(* Logix 5000 project; controller TBEN_Lx_8IOL_AOI_V0_2 vendor 1 type 14 code 176 rev 32.11; software revision 32.00; part 5 of 16 *)

           TBEN_L4_8IOL:O.Data[63].0   // IO-Link Port 4 - Output data word 13 (INT bit0)
           TBEN_L4_8IOL:O.Data[63].1   // IO-Link Port 4 - Output data word 13 (INT bit1)
           TBEN_L4_8IOL:O.Data[63].10   // IO-Link Port 4 - Output data word 13 (INT bit10)
           TBEN_L4_8IOL:O.Data[63].11   // IO-Link Port 4 - Output data word 13 (INT bit11)
           TBEN_L4_8IOL:O.Data[63].12   // IO-Link Port 4 - Output data word 13 (INT bit12)
           TBEN_L4_8IOL:O.Data[63].13   // IO-Link Port 4 - Output data word 13 (INT bit13)
           TBEN_L4_8IOL:O.Data[63].14   // IO-Link Port 4 - Output data word 13 (INT bit14)
           TBEN_L4_8IOL:O.Data[63].15   // IO-Link Port 4 - Output data word 13 (INT bit15)
           TBEN_L4_8IOL:O.Data[63].2   // IO-Link Port 4 - Output data word 13 (INT bit2)
           TBEN_L4_8IOL:O.Data[63].3   // IO-Link Port 4 - Output data word 13 (INT bit3)
           TBEN_L4_8IOL:O.Data[63].4   // IO-Link Port 4 - Output data word 13 (INT bit4)
           TBEN_L4_8IOL:O.Data[63].5   // IO-Link Port 4 - Output data word 13 (INT bit5)
           TBEN_L4_8IOL:O.Data[63].6   // IO-Link Port 4 - Output data word 13 (INT bit6)
           TBEN_L4_8IOL:O.Data[63].7   // IO-Link Port 4 - Output data word 13 (INT bit7)
           TBEN_L4_8IOL:O.Data[63].8   // IO-Link Port 4 - Output data word 13 (INT bit8)
           TBEN_L4_8IOL:O.Data[63].9   // IO-Link Port 4 - Output data word 13 (INT bit9)
           TBEN_L4_8IOL:O.Data[64]   // IO-Link Port 4 - Output data word 14
           TBEN_L4_8IOL:O.Data[64].0   // IO-Link Port 4 - Output data word 14 (INT bit0)
           TBEN_L4_8IOL:O.Data[64].1   // IO-Link Port 4 - Output data word 14 (INT bit1)
           TBEN_L4_8IOL:O.Data[64].10   // IO-Link Port 4 - Output data word 14 (INT bit10)
           TBEN_L4_8IOL:O.Data[64].11   // IO-Link Port 4 - Output data word 14 (INT bit11)
           TBEN_L4_8IOL:O.Data[64].12   // IO-Link Port 4 - Output data word 14 (INT bit12)
           TBEN_L4_8IOL:O.Data[64].13   // IO-Link Port 4 - Output data word 14 (INT bit13)
           TBEN_L4_8IOL:O.Data[64].14   // IO-Link Port 4 - Output data word 14 (INT bit14)
           TBEN_L4_8IOL:O.Data[64].15   // IO-Link Port 4 - Output data word 14 (INT bit15)
           TBEN_L4_8IOL:O.Data[64].2   // IO-Link Port 4 - Output data word 14 (INT bit2)
           TBEN_L4_8IOL:O.Data[64].3   // IO-Link Port 4 - Output data word 14 (INT bit3)
           TBEN_L4_8IOL:O.Data[64].4   // IO-Link Port 4 - Output data word 14 (INT bit4)
           TBEN_L4_8IOL:O.Data[64].5   // IO-Link Port 4 - Output data word 14 (INT bit5)
           TBEN_L4_8IOL:O.Data[64].6   // IO-Link Port 4 - Output data word 14 (INT bit6)
           TBEN_L4_8IOL:O.Data[64].7   // IO-Link Port 4 - Output data word 14 (INT bit7)
           TBEN_L4_8IOL:O.Data[64].8   // IO-Link Port 4 - Output data word 14 (INT bit8)
           TBEN_L4_8IOL:O.Data[64].9   // IO-Link Port 4 - Output data word 14 (INT bit9)
           TBEN_L4_8IOL:O.Data[65]   // IO-Link Port 4 - Output data word 15
           TBEN_L4_8IOL:O.Data[65].0   // IO-Link Port 4 - Output data word 15 (INT bit0)
           TBEN_L4_8IOL:O.Data[65].1   // IO-Link Port 4 - Output data word 15 (INT bit1)
           TBEN_L4_8IOL:O.Data[65].10   // IO-Link Port 4 - Output data word 15 (INT bit10)
           TBEN_L4_8IOL:O.Data[65].11   // IO-Link Port 4 - Output data word 15 (INT bit11)
           TBEN_L4_8IOL:O.Data[65].12   // IO-Link Port 4 - Output data word 15 (INT bit12)
           TBEN_L4_8IOL:O.Data[65].13   // IO-Link Port 4 - Output data word 15 (INT bit13)
           TBEN_L4_8IOL:O.Data[65].14   // IO-Link Port 4 - Output data word 15 (INT bit14)
           TBEN_L4_8IOL:O.Data[65].15   // IO-Link Port 4 - Output data word 15 (INT bit15)
           TBEN_L4_8IOL:O.Data[65].2   // IO-Link Port 4 - Output data word 15 (INT bit2)
           TBEN_L4_8IOL:O.Data[65].3   // IO-Link Port 4 - Output data word 15 (INT bit3)
           TBEN_L4_8IOL:O.Data[65].4   // IO-Link Port 4 - Output data word 15 (INT bit4)
           TBEN_L4_8IOL:O.Data[65].5   // IO-Link Port 4 - Output data word 15 (INT bit5)
           TBEN_L4_8IOL:O.Data[65].6   // IO-Link Port 4 - Output data word 15 (INT bit6)
           TBEN_L4_8IOL:O.Data[65].7   // IO-Link Port 4 - Output data word 15 (INT bit7)
           TBEN_L4_8IOL:O.Data[65].8   // IO-Link Port 4 - Output data word 15 (INT bit8)
           TBEN_L4_8IOL:O.Data[65].9   // IO-Link Port 4 - Output data word 15 (INT bit9)
           TBEN_L4_8IOL:O.Data[66]   // IO-Link Port 5 - Output data word 0
           TBEN_L4_8IOL:O.Data[66].0   // IO-Link Port 5 - Output data word 0 (INT bit0)
           TBEN_L4_8IOL:O.Data[66].1   // IO-Link Port 5 - Output data word 0 (INT bit1)
           TBEN_L4_8IOL:O.Data[66].10   // IO-Link Port 5 - Output data word 0 (INT bit10)
           TBEN_L4_8IOL:O.Data[66].11   // IO-Link Port 5 - Output data word 0 (INT bit11)
           TBEN_L4_8IOL:O.Data[66].12   // IO-Link Port 5 - Output data word 0 (INT bit12)
           TBEN_L4_8IOL:O.Data[66].13   // IO-Link Port 5 - Output data word 0 (INT bit13)
           TBEN_L4_8IOL:O.Data[66].14   // IO-Link Port 5 - Output data word 0 (INT bit14)
           TBEN_L4_8IOL:O.Data[66].15   // IO-Link Port 5 - Output data word 0 (INT bit15)
           TBEN_L4_8IOL:O.Data[66].2   // IO-Link Port 5 - Output data word 0 (INT bit2)
           TBEN_L4_8IOL:O.Data[66].3   // IO-Link Port 5 - Output data word 0 (INT bit3)
           TBEN_L4_8IOL:O.Data[66].4   // IO-Link Port 5 - Output data word 0 (INT bit4)
           TBEN_L4_8IOL:O.Data[66].5   // IO-Link Port 5 - Output data word 0 (INT bit5)
           TBEN_L4_8IOL:O.Data[66].6   // IO-Link Port 5 - Output data word 0 (INT bit6)
           TBEN_L4_8IOL:O.Data[66].7   // IO-Link Port 5 - Output data word 0 (INT bit7)
           TBEN_L4_8IOL:O.Data[66].8   // IO-Link Port 5 - Output data word 0 (INT bit8)
           TBEN_L4_8IOL:O.Data[66].9   // IO-Link Port 5 - Output data word 0 (INT bit9)
           TBEN_L4_8IOL:O.Data[67]   // IO-Link Port 5 - Output data word 1
           TBEN_L4_8IOL:O.Data[67].0   // IO-Link Port 5 - Output data word 1 (INT bit0)
           TBEN_L4_8IOL:O.Data[67].1   // IO-Link Port 5 - Output data word 1 (INT bit1)
           TBEN_L4_8IOL:O.Data[67].10   // IO-Link Port 5 - Output data word 1 (INT bit10)
           TBEN_L4_8IOL:O.Data[67].11   // IO-Link Port 5 - Output data word 1 (INT bit11)
           TBEN_L4_8IOL:O.Data[67].12   // IO-Link Port 5 - Output data word 1 (INT bit12)
           TBEN_L4_8IOL:O.Data[67].13   // IO-Link Port 5 - Output data word 1 (INT bit13)
           TBEN_L4_8IOL:O.Data[67].14   // IO-Link Port 5 - Output data word 1 (INT bit14)
           TBEN_L4_8IOL:O.Data[67].15   // IO-Link Port 5 - Output data word 1 (INT bit15)
           TBEN_L4_8IOL:O.Data[67].2   // IO-Link Port 5 - Output data word 1 (INT bit2)
           TBEN_L4_8IOL:O.Data[67].3   // IO-Link Port 5 - Output data word 1 (INT bit3)
           TBEN_L4_8IOL:O.Data[67].4   // IO-Link Port 5 - Output data word 1 (INT bit4)
           TBEN_L4_8IOL:O.Data[67].5   // IO-Link Port 5 - Output data word 1 (INT bit5)
           TBEN_L4_8IOL:O.Data[67].6   // IO-Link Port 5 - Output data word 1 (INT bit6)
           TBEN_L4_8IOL:O.Data[67].7   // IO-Link Port 5 - Output data word 1 (INT bit7)
           TBEN_L4_8IOL:O.Data[67].8   // IO-Link Port 5 - Output data word 1 (INT bit8)
           TBEN_L4_8IOL:O.Data[67].9   // IO-Link Port 5 - Output data word 1 (INT bit9)
           TBEN_L4_8IOL:O.Data[68]   // IO-Link Port 5 - Output data word 2
           TBEN_L4_8IOL:O.Data[68].0   // IO-Link Port 5 - Output data word 2 (INT bit0)
           TBEN_L4_8IOL:O.Data[68].1   // IO-Link Port 5 - Output data word 2 (INT bit1)
           TBEN_L4_8IOL:O.Data[68].10   // IO-Link Port 5 - Output data word 2 (INT bit10)
           TBEN_L4_8IOL:O.Data[68].11   // IO-Link Port 5 - Output data word 2 (INT bit11)
           TBEN_L4_8IOL:O.Data[68].12   // IO-Link Port 5 - Output data word 2 (INT bit12)
           TBEN_L4_8IOL:O.Data[68].13   // IO-Link Port 5 - Output data word 2 (INT bit13)
           TBEN_L4_8IOL:O.Data[68].14   // IO-Link Port 5 - Output data word 2 (INT bit14)
           TBEN_L4_8IOL:O.Data[68].15   // IO-Link Port 5 - Output data word 2 (INT bit15)
           TBEN_L4_8IOL:O.Data[68].2   // IO-Link Port 5 - Output data word 2 (INT bit2)
           TBEN_L4_8IOL:O.Data[68].3   // IO-Link Port 5 - Output data word 2 (INT bit3)
           TBEN_L4_8IOL:O.Data[68].4   // IO-Link Port 5 - Output data word 2 (INT bit4)
           TBEN_L4_8IOL:O.Data[68].5   // IO-Link Port 5 - Output data word 2 (INT bit5)
           TBEN_L4_8IOL:O.Data[68].6   // IO-Link Port 5 - Output data word 2 (INT bit6)
           TBEN_L4_8IOL:O.Data[68].7   // IO-Link Port 5 - Output data word 2 (INT bit7)
           TBEN_L4_8IOL:O.Data[68].8   // IO-Link Port 5 - Output data word 2 (INT bit8)
           TBEN_L4_8IOL:O.Data[68].9   // IO-Link Port 5 - Output data word 2 (INT bit9)
           TBEN_L4_8IOL:O.Data[69]   // IO-Link Port 5 - Output data word 3
           TBEN_L4_8IOL:O.Data[69].0   // IO-Link Port 5 - Output data word 3 (INT bit0)
           TBEN_L4_8IOL:O.Data[69].1   // IO-Link Port 5 - Output data word 3 (INT bit1)
           TBEN_L4_8IOL:O.Data[69].10   // IO-Link Port 5 - Output data word 3 (INT bit10)
           TBEN_L4_8IOL:O.Data[69].11   // IO-Link Port 5 - Output data word 3 (INT bit11)
           TBEN_L4_8IOL:O.Data[69].12   // IO-Link Port 5 - Output data word 3 (INT bit12)
           TBEN_L4_8IOL:O.Data[69].13   // IO-Link Port 5 - Output data word 3 (INT bit13)
           TBEN_L4_8IOL:O.Data[69].14   // IO-Link Port 5 - Output data word 3 (INT bit14)
           TBEN_L4_8IOL:O.Data[69].15   // IO-Link Port 5 - Output data word 3 (INT bit15)
           TBEN_L4_8IOL:O.Data[69].2   // IO-Link Port 5 - Output data word 3 (INT bit2)
           TBEN_L4_8IOL:O.Data[69].3   // IO-Link Port 5 - Output data word 3 (INT bit3)
           TBEN_L4_8IOL:O.Data[69].4   // IO-Link Port 5 - Output data word 3 (INT bit4)
           TBEN_L4_8IOL:O.Data[69].5   // IO-Link Port 5 - Output data word 3 (INT bit5)
           TBEN_L4_8IOL:O.Data[69].6   // IO-Link Port 5 - Output data word 3 (INT bit6)
           TBEN_L4_8IOL:O.Data[69].7   // IO-Link Port 5 - Output data word 3 (INT bit7)
           TBEN_L4_8IOL:O.Data[69].8   // IO-Link Port 5 - Output data word 3 (INT bit8)
           TBEN_L4_8IOL:O.Data[69].9   // IO-Link Port 5 - Output data word 3 (INT bit9)
           TBEN_L4_8IOL:O.Data[6]   // IO-Link Port 1 - Output data word 4
           TBEN_L4_8IOL:O.Data[6].0   // IO-Link Port 1 - Output data word 4 (INT bit0)
           TBEN_L4_8IOL:O.Data[6].1   // IO-Link Port 1 - Output data word 4 (INT bit1)
           TBEN_L4_8IOL:O.Data[6].10   // IO-Link Port 1 - Output data word 4 (INT bit10)
           TBEN_L4_8IOL:O.Data[6].11   // IO-Link Port 1 - Output data word 4 (INT bit11)
           TBEN_L4_8IOL:O.Data[6].12   // IO-Link Port 1 - Output data word 4 (INT bit12)
           TBEN_L4_8IOL:O.Data[6].13   // IO-Link Port 1 - Output data word 4 (INT bit13)
           TBEN_L4_8IOL:O.Data[6].14   // IO-Link Port 1 - Output data word 4 (INT bit14)
           TBEN_L4_8IOL:O.Data[6].15   // IO-Link Port 1 - Output data word 4 (INT bit15)
           TBEN_L4_8IOL:O.Data[6].2   // IO-Link Port 1 - Output data word 4 (INT bit2)
           TBEN_L4_8IOL:O.Data[6].3   // IO-Link Port 1 - Output data word 4 (INT bit3)
           TBEN_L4_8IOL:O.Data[6].4   // IO-Link Port 1 - Output data word 4 (INT bit4)
           TBEN_L4_8IOL:O.Data[6].5   // IO-Link Port 1 - Output data word 4 (INT bit5)
           TBEN_L4_8IOL:O.Data[6].6   // IO-Link Port 1 - Output data word 4 (INT bit6)
           TBEN_L4_8IOL:O.Data[6].7   // IO-Link Port 1 - Output data word 4 (INT bit7)
           TBEN_L4_8IOL:O.Data[6].8   // IO-Link Port 1 - Output data word 4 (INT bit8)
           TBEN_L4_8IOL:O.Data[6].9   // IO-Link Port 1 - Output data word 4 (INT bit9)
           TBEN_L4_8IOL:O.Data[70]   // IO-Link Port 5 - Output data word 4
           TBEN_L4_8IOL:O.Data[70].0   // IO-Link Port 5 - Output data word 4 (INT bit0)
           TBEN_L4_8IOL:O.Data[70].1   // IO-Link Port 5 - Output data word 4 (INT bit1)
           TBEN_L4_8IOL:O.Data[70].10   // IO-Link Port 5 - Output data word 4 (INT bit10)
           TBEN_L4_8IOL:O.Data[70].11   // IO-Link Port 5 - Output data word 4 (INT bit11)
           TBEN_L4_8IOL:O.Data[70].12   // IO-Link Port 5 - Output data word 4 (INT bit12)
           TBEN_L4_8IOL:O.Data[70].13   // IO-Link Port 5 - Output data word 4 (INT bit13)
           TBEN_L4_8IOL:O.Data[70].14   // IO-Link Port 5 - Output data word 4 (INT bit14)
           TBEN_L4_8IOL:O.Data[70].15   // IO-Link Port 5 - Output data word 4 (INT bit15)
           TBEN_L4_8IOL:O.Data[70].2   // IO-Link Port 5 - Output data word 4 (INT bit2)
           TBEN_L4_8IOL:O.Data[70].3   // IO-Link Port 5 - Output data word 4 (INT bit3)
           TBEN_L4_8IOL:O.Data[70].4   // IO-Link Port 5 - Output data word 4 (INT bit4)
           TBEN_L4_8IOL:O.Data[70].5   // IO-Link Port 5 - Output data word 4 (INT bit5)
           TBEN_L4_8IOL:O.Data[70].6   // IO-Link Port 5 - Output data word 4 (INT bit6)
           TBEN_L4_8IOL:O.Data[70].7   // IO-Link Port 5 - Output data word 4 (INT bit7)
           TBEN_L4_8IOL:O.Data[70].8   // IO-Link Port 5 - Output data word 4 (INT bit8)
           TBEN_L4_8IOL:O.Data[70].9   // IO-Link Port 5 - Output data word 4 (INT bit9)
           TBEN_L4_8IOL:O.Data[71]   // IO-Link Port 5 - Output data word 5
           TBEN_L4_8IOL:O.Data[71].0   // IO-Link Port 5 - Output data word 5 (INT bit0)
           TBEN_L4_8IOL:O.Data[71].1   // IO-Link Port 5 - Output data word 5 (INT bit1)
           TBEN_L4_8IOL:O.Data[71].10   // IO-Link Port 5 - Output data word 5 (INT bit10)
           TBEN_L4_8IOL:O.Data[71].11   // IO-Link Port 5 - Output data word 5 (INT bit11)
           TBEN_L4_8IOL:O.Data[71].12   // IO-Link Port 5 - Output data word 5 (INT bit12)
           TBEN_L4_8IOL:O.Data[71].13   // IO-Link Port 5 - Output data word 5 (INT bit13)
           TBEN_L4_8IOL:O.Data[71].14   // IO-Link Port 5 - Output data word 5 (INT bit14)
           TBEN_L4_8IOL:O.Data[71].15   // IO-Link Port 5 - Output data word 5 (INT bit15)
           TBEN_L4_8IOL:O.Data[71].2   // IO-Link Port 5 - Output data word 5 (INT bit2)
           TBEN_L4_8IOL:O.Data[71].3   // IO-Link Port 5 - Output data word 5 (INT bit3)
           TBEN_L4_8IOL:O.Data[71].4   // IO-Link Port 5 - Output data word 5 (INT bit4)
           TBEN_L4_8IOL:O.Data[71].5   // IO-Link Port 5 - Output data word 5 (INT bit5)
           TBEN_L4_8IOL:O.Data[71].6   // IO-Link Port 5 - Output data word 5 (INT bit6)
           TBEN_L4_8IOL:O.Data[71].7   // IO-Link Port 5 - Output data word 5 (INT bit7)
           TBEN_L4_8IOL:O.Data[71].8   // IO-Link Port 5 - Output data word 5 (INT bit8)
           TBEN_L4_8IOL:O.Data[71].9   // IO-Link Port 5 - Output data word 5 (INT bit9)
           TBEN_L4_8IOL:O.Data[72]   // IO-Link Port 5 - Output data word 6
           TBEN_L4_8IOL:O.Data[72].0   // IO-Link Port 5 - Output data word 6 (INT bit0)
           TBEN_L4_8IOL:O.Data[72].1   // IO-Link Port 5 - Output data word 6 (INT bit1)
           TBEN_L4_8IOL:O.Data[72].10   // IO-Link Port 5 - Output data word 6 (INT bit10)
           TBEN_L4_8IOL:O.Data[72].11   // IO-Link Port 5 - Output data word 6 (INT bit11)
           TBEN_L4_8IOL:O.Data[72].12   // IO-Link Port 5 - Output data word 6 (INT bit12)
           TBEN_L4_8IOL:O.Data[72].13   // IO-Link Port 5 - Output data word 6 (INT bit13)
           TBEN_L4_8IOL:O.Data[72].14   // IO-Link Port 5 - Output data word 6 (INT bit14)
           TBEN_L4_8IOL:O.Data[72].15   // IO-Link Port 5 - Output data word 6 (INT bit15)
           TBEN_L4_8IOL:O.Data[72].2   // IO-Link Port 5 - Output data word 6 (INT bit2)
           TBEN_L4_8IOL:O.Data[72].3   // IO-Link Port 5 - Output data word 6 (INT bit3)
           TBEN_L4_8IOL:O.Data[72].4   // IO-Link Port 5 - Output data word 6 (INT bit4)
           TBEN_L4_8IOL:O.Data[72].5   // IO-Link Port 5 - Output data word 6 (INT bit5)
           TBEN_L4_8IOL:O.Data[72].6   // IO-Link Port 5 - Output data word 6 (INT bit6)
           TBEN_L4_8IOL:O.Data[72].7   // IO-Link Port 5 - Output data word 6 (INT bit7)
           TBEN_L4_8IOL:O.Data[72].8   // IO-Link Port 5 - Output data word 6 (INT bit8)
           TBEN_L4_8IOL:O.Data[72].9   // IO-Link Port 5 - Output data word 6 (INT bit9)
           TBEN_L4_8IOL:O.Data[73]   // IO-Link Port 5 - Output data word 7
           TBEN_L4_8IOL:O.Data[73].0   // IO-Link Port 5 - Output data word 7 (INT bit0)
           TBEN_L4_8IOL:O.Data[73].1   // IO-Link Port 5 - Output data word 7 (INT bit1)
           TBEN_L4_8IOL:O.Data[73].10   // IO-Link Port 5 - Output data word 7 (INT bit10)
           TBEN_L4_8IOL:O.Data[73].11   // IO-Link Port 5 - Output data word 7 (INT bit11)
           TBEN_L4_8IOL:O.Data[73].12   // IO-Link Port 5 - Output data word 7 (INT bit12)
           TBEN_L4_8IOL:O.Data[73].13   // IO-Link Port 5 - Output data word 7 (INT bit13)
           TBEN_L4_8IOL:O.Data[73].14   // IO-Link Port 5 - Output data word 7 (INT bit14)
           TBEN_L4_8IOL:O.Data[73].15   // IO-Link Port 5 - Output data word 7 (INT bit15)
           TBEN_L4_8IOL:O.Data[73].2   // IO-Link Port 5 - Output data word 7 (INT bit2)
           TBEN_L4_8IOL:O.Data[73].3   // IO-Link Port 5 - Output data word 7 (INT bit3)
           TBEN_L4_8IOL:O.Data[73].4   // IO-Link Port 5 - Output data word 7 (INT bit4)
           TBEN_L4_8IOL:O.Data[73].5   // IO-Link Port 5 - Output data word 7 (INT bit5)
           TBEN_L4_8IOL:O.Data[73].6   // IO-Link Port 5 - Output data word 7 (INT bit6)
           TBEN_L4_8IOL:O.Data[73].7   // IO-Link Port 5 - Output data word 7 (INT bit7)
           TBEN_L4_8IOL:O.Data[73].8   // IO-Link Port 5 - Output data word 7 (INT bit8)
           TBEN_L4_8IOL:O.Data[73].9   // IO-Link Port 5 - Output data word 7 (INT bit9)
           TBEN_L4_8IOL:O.Data[74]   // IO-Link Port 5 - Output data word 8
           TBEN_L4_8IOL:O.Data[74].0   // IO-Link Port 5 - Output data word 8 (INT bit0)
           TBEN_L4_8IOL:O.Data[74].1   // IO-Link Port 5 - Output data word 8 (INT bit1)
           TBEN_L4_8IOL:O.Data[74].10   // IO-Link Port 5 - Output data word 8 (INT bit10)
           TBEN_L4_8IOL:O.Data[74].11   // IO-Link Port 5 - Output data word 8 (INT bit11)
           TBEN_L4_8IOL:O.Data[74].12   // IO-Link Port 5 - Output data word 8 (INT bit12)
           TBEN_L4_8IOL:O.Data[74].13   // IO-Link Port 5 - Output data word 8 (INT bit13)
           TBEN_L4_8IOL:O.Data[74].14   // IO-Link Port 5 - Output data word 8 (INT bit14)
           TBEN_L4_8IOL:O.Data[74].15   // IO-Link Port 5 - Output data word 8 (INT bit15)
           TBEN_L4_8IOL:O.Data[74].2   // IO-Link Port 5 - Output data word 8 (INT bit2)
           TBEN_L4_8IOL:O.Data[74].3   // IO-Link Port 5 - Output data word 8 (INT bit3)
           TBEN_L4_8IOL:O.Data[74].4   // IO-Link Port 5 - Output data word 8 (INT bit4)
           TBEN_L4_8IOL:O.Data[74].5   // IO-Link Port 5 - Output data word 8 (INT bit5)
           TBEN_L4_8IOL:O.Data[74].6   // IO-Link Port 5 - Output data word 8 (INT bit6)
           TBEN_L4_8IOL:O.Data[74].7   // IO-Link Port 5 - Output data word 8 (INT bit7)
           TBEN_L4_8IOL:O.Data[74].8   // IO-Link Port 5 - Output data word 8 (INT bit8)
           TBEN_L4_8IOL:O.Data[74].9   // IO-Link Port 5 - Output data word 8 (INT bit9)
           TBEN_L4_8IOL:O.Data[75]   // IO-Link Port 5 - Output data word 9
           TBEN_L4_8IOL:O.Data[75].0   // IO-Link Port 5 - Output data word 9 (INT bit0)
           TBEN_L4_8IOL:O.Data[75].1   // IO-Link Port 5 - Output data word 9 (INT bit1)
           TBEN_L4_8IOL:O.Data[75].10   // IO-Link Port 5 - Output data word 9 (INT bit10)
           TBEN_L4_8IOL:O.Data[75].11   // IO-Link Port 5 - Output data word 9 (INT bit11)
           TBEN_L4_8IOL:O.Data[75].12   // IO-Link Port 5 - Output data word 9 (INT bit12)
           TBEN_L4_8IOL:O.Data[75].13   // IO-Link Port 5 - Output data word 9 (INT bit13)
           TBEN_L4_8IOL:O.Data[75].14   // IO-Link Port 5 - Output data word 9 (INT bit14)
           TBEN_L4_8IOL:O.Data[75].15   // IO-Link Port 5 - Output data word 9 (INT bit15)
           TBEN_L4_8IOL:O.Data[75].2   // IO-Link Port 5 - Output data word 9 (INT bit2)
           TBEN_L4_8IOL:O.Data[75].3   // IO-Link Port 5 - Output data word 9 (INT bit3)
           TBEN_L4_8IOL:O.Data[75].4   // IO-Link Port 5 - Output data word 9 (INT bit4)
           TBEN_L4_8IOL:O.Data[75].5   // IO-Link Port 5 - Output data word 9 (INT bit5)
           TBEN_L4_8IOL:O.Data[75].6   // IO-Link Port 5 - Output data word 9 (INT bit6)
           TBEN_L4_8IOL:O.Data[75].7   // IO-Link Port 5 - Output data word 9 (INT bit7)
           TBEN_L4_8IOL:O.Data[75].8   // IO-Link Port 5 - Output data word 9 (INT bit8)
           TBEN_L4_8IOL:O.Data[75].9   // IO-Link Port 5 - Output data word 9 (INT bit9)
           TBEN_L4_8IOL:O.Data[76]   // IO-Link Port 5 - Output data word 10
           TBEN_L4_8IOL:O.Data[76].0   // IO-Link Port 5 - Output data word 10 (INT bit0)
           TBEN_L4_8IOL:O.Data[76].1   // IO-Link Port 5 - Output data word 10 (INT bit1)
           TBEN_L4_8IOL:O.Data[76].10   // IO-Link Port 5 - Output data word 10 (INT bit10)
           TBEN_L4_8IOL:O.Data[76].11   // IO-Link Port 5 - Output data word 10 (INT bit11)
           TBEN_L4_8IOL:O.Data[76].12   // IO-Link Port 5 - Output data word 10 (INT bit12)
           TBEN_L4_8IOL:O.Data[76].13   // IO-Link Port 5 - Output data word 10 (INT bit13)
           TBEN_L4_8IOL:O.Data[76].14   // IO-Link Port 5 - Output data word 10 (INT bit14)
           TBEN_L4_8IOL:O.Data[76].15   // IO-Link Port 5 - Output data word 10 (INT bit15)
           TBEN_L4_8IOL:O.Data[76].2   // IO-Link Port 5 - Output data word 10 (INT bit2)
           TBEN_L4_8IOL:O.Data[76].3   // IO-Link Port 5 - Output data word 10 (INT bit3)
           TBEN_L4_8IOL:O.Data[76].4   // IO-Link Port 5 - Output data word 10 (INT bit4)
           TBEN_L4_8IOL:O.Data[76].5   // IO-Link Port 5 - Output data word 10 (INT bit5)
           TBEN_L4_8IOL:O.Data[76].6   // IO-Link Port 5 - Output data word 10 (INT bit6)
           TBEN_L4_8IOL:O.Data[76].7   // IO-Link Port 5 - Output data word 10 (INT bit7)
           TBEN_L4_8IOL:O.Data[76].8   // IO-Link Port 5 - Output data word 10 (INT bit8)
           TBEN_L4_8IOL:O.Data[76].9   // IO-Link Port 5 - Output data word 10 (INT bit9)
           TBEN_L4_8IOL:O.Data[77]   // IO-Link Port 5 - Output data word 11
           TBEN_L4_8IOL:O.Data[77].0   // IO-Link Port 5 - Output data word 11 (INT bit0)
           TBEN_L4_8IOL:O.Data[77].1   // IO-Link Port 5 - Output data word 11 (INT bit1)
           TBEN_L4_8IOL:O.Data[77].10   // IO-Link Port 5 - Output data word 11 (INT bit10)
           TBEN_L4_8IOL:O.Data[77].11   // IO-Link Port 5 - Output data word 11 (INT bit11)
           TBEN_L4_8IOL:O.Data[77].12   // IO-Link Port 5 - Output data word 11 (INT bit12)
           TBEN_L4_8IOL:O.Data[77].13   // IO-Link Port 5 - Output data word 11 (INT bit13)
           TBEN_L4_8IOL:O.Data[77].14   // IO-Link Port 5 - Output data word 11 (INT bit14)
           TBEN_L4_8IOL:O.Data[77].15   // IO-Link Port 5 - Output data word 11 (INT bit15)
           TBEN_L4_8IOL:O.Data[77].2   // IO-Link Port 5 - Output data word 11 (INT bit2)
           TBEN_L4_8IOL:O.Data[77].3   // IO-Link Port 5 - Output data word 11 (INT bit3)
           TBEN_L4_8IOL:O.Data[77].4   // IO-Link Port 5 - Output data word 11 (INT bit4)
           TBEN_L4_8IOL:O.Data[77].5   // IO-Link Port 5 - Output data word 11 (INT bit5)
           TBEN_L4_8IOL:O.Data[77].6   // IO-Link Port 5 - Output data word 11 (INT bit6)
           TBEN_L4_8IOL:O.Data[77].7   // IO-Link Port 5 - Output data word 11 (INT bit7)
           TBEN_L4_8IOL:O.Data[77].8   // IO-Link Port 5 - Output data word 11 (INT bit8)
           TBEN_L4_8IOL:O.Data[77].9   // IO-Link Port 5 - Output data word 11 (INT bit9)
           TBEN_L4_8IOL:O.Data[78]   // IO-Link Port 5 - Output data word 12
           TBEN_L4_8IOL:O.Data[78].0   // IO-Link Port 5 - Output data word 12 (INT bit0)
           TBEN_L4_8IOL:O.Data[78].1   // IO-Link Port 5 - Output data word 12 (INT bit1)
           TBEN_L4_8IOL:O.Data[78].10   // IO-Link Port 5 - Output data word 12 (INT bit10)
           TBEN_L4_8IOL:O.Data[78].11   // IO-Link Port 5 - Output data word 12 (INT bit11)
           TBEN_L4_8IOL:O.Data[78].12   // IO-Link Port 5 - Output data word 12 (INT bit12)
           TBEN_L4_8IOL:O.Data[78].13   // IO-Link Port 5 - Output data word 12 (INT bit13)
           TBEN_L4_8IOL:O.Data[78].14   // IO-Link Port 5 - Output data word 12 (INT bit14)
           TBEN_L4_8IOL:O.Data[78].15   // IO-Link Port 5 - Output data word 12 (INT bit15)
           TBEN_L4_8IOL:O.Data[78].2   // IO-Link Port 5 - Output data word 12 (INT bit2)
           TBEN_L4_8IOL:O.Data[78].3   // IO-Link Port 5 - Output data word 12 (INT bit3)
           TBEN_L4_8IOL:O.Data[78].4   // IO-Link Port 5 - Output data word 12 (INT bit4)
           TBEN_L4_8IOL:O.Data[78].5   // IO-Link Port 5 - Output data word 12 (INT bit5)
           TBEN_L4_8IOL:O.Data[78].6   // IO-Link Port 5 - Output data word 12 (INT bit6)
           TBEN_L4_8IOL:O.Data[78].7   // IO-Link Port 5 - Output data word 12 (INT bit7)
           TBEN_L4_8IOL:O.Data[78].8   // IO-Link Port 5 - Output data word 12 (INT bit8)
           TBEN_L4_8IOL:O.Data[78].9   // IO-Link Port 5 - Output data word 12 (INT bit9)
           TBEN_L4_8IOL:O.Data[79]   // IO-Link Port 5 - Output data word 13
           TBEN_L4_8IOL:O.Data[79].0   // IO-Link Port 5 - Output data word 13 (INT bit0)
           TBEN_L4_8IOL:O.Data[79].1   // IO-Link Port 5 - Output data word 13 (INT bit1)
           TBEN_L4_8IOL:O.Data[79].10   // IO-Link Port 5 - Output data word 13 (INT bit10)
           TBEN_L4_8IOL:O.Data[79].11   // IO-Link Port 5 - Output data word 13 (INT bit11)
           TBEN_L4_8IOL:O.Data[79].12   // IO-Link Port 5 - Output data word 13 (INT bit12)
           TBEN_L4_8IOL:O.Data[79].13   // IO-Link Port 5 - Output data word 13 (INT bit13)
           TBEN_L4_8IOL:O.Data[79].14   // IO-Link Port 5 - Output data word 13 (INT bit14)
           TBEN_L4_8IOL:O.Data[79].15   // IO-Link Port 5 - Output data word 13 (INT bit15)
           TBEN_L4_8IOL:O.Data[79].2   // IO-Link Port 5 - Output data word 13 (INT bit2)
           TBEN_L4_8IOL:O.Data[79].3   // IO-Link Port 5 - Output data word 13 (INT bit3)
           TBEN_L4_8IOL:O.Data[79].4   // IO-Link Port 5 - Output data word 13 (INT bit4)
           TBEN_L4_8IOL:O.Data[79].5   // IO-Link Port 5 - Output data word 13 (INT bit5)
           TBEN_L4_8IOL:O.Data[79].6   // IO-Link Port 5 - Output data word 13 (INT bit6)
           TBEN_L4_8IOL:O.Data[79].7   // IO-Link Port 5 - Output data word 13 (INT bit7)
           TBEN_L4_8IOL:O.Data[79].8   // IO-Link Port 5 - Output data word 13 (INT bit8)
           TBEN_L4_8IOL:O.Data[79].9   // IO-Link Port 5 - Output data word 13 (INT bit9)
           TBEN_L4_8IOL:O.Data[7]   // IO-Link Port 1 - Output data word 5
           TBEN_L4_8IOL:O.Data[7].0   // IO-Link Port 1 - Output data word 5 (INT bit0)
           TBEN_L4_8IOL:O.Data[7].1   // IO-Link Port 1 - Output data word 5 (INT bit1)
           TBEN_L4_8IOL:O.Data[7].10   // IO-Link Port 1 - Output data word 5 (INT bit10)
           TBEN_L4_8IOL:O.Data[7].11   // IO-Link Port 1 - Output data word 5 (INT bit11)
           TBEN_L4_8IOL:O.Data[7].12   // IO-Link Port 1 - Output data word 5 (INT bit12)
           TBEN_L4_8IOL:O.Data[7].13   // IO-Link Port 1 - Output data word 5 (INT bit13)
           TBEN_L4_8IOL:O.Data[7].14   // IO-Link Port 1 - Output data word 5 (INT bit14)
           TBEN_L4_8IOL:O.Data[7].15   // IO-Link Port 1 - Output data word 5 (INT bit15)
           TBEN_L4_8IOL:O.Data[7].2   // IO-Link Port 1 - Output data word 5 (INT bit2)
           TBEN_L4_8IOL:O.Data[7].3   // IO-Link Port 1 - Output data word 5 (INT bit3)
           TBEN_L4_8IOL:O.Data[7].4   // IO-Link Port 1 - Output data word 5 (INT bit4)
           TBEN_L4_8IOL:O.Data[7].5   // IO-Link Port 1 - Output data word 5 (INT bit5)
           TBEN_L4_8IOL:O.Data[7].6   // IO-Link Port 1 - Output data word 5 (INT bit6)
           TBEN_L4_8IOL:O.Data[7].7   // IO-Link Port 1 - Output data word 5 (INT bit7)
           TBEN_L4_8IOL:O.Data[7].8   // IO-Link Port 1 - Output data word 5 (INT bit8)
           TBEN_L4_8IOL:O.Data[7].9   // IO-Link Port 1 - Output data word 5 (INT bit9)
           TBEN_L4_8IOL:O.Data[80]   // IO-Link Port 5 - Output data word 14
           TBEN_L4_8IOL:O.Data[80].0   // IO-Link Port 5 - Output data word 14 (INT bit0)
           TBEN_L4_8IOL:O.Data[80].1   // IO-Link Port 5 - Output data word 14 (INT bit1)
           TBEN_L4_8IOL:O.Data[80].10   // IO-Link Port 5 - Output data word 14 (INT bit10)
           TBEN_L4_8IOL:O.Data[80].11   // IO-Link Port 5 - Output data word 14 (INT bit11)
           TBEN_L4_8IOL:O.Data[80].12   // IO-Link Port 5 - Output data word 14 (INT bit12)
           TBEN_L4_8IOL:O.Data[80].13   // IO-Link Port 5 - Output data word 14 (INT bit13)
           TBEN_L4_8IOL:O.Data[80].14   // IO-Link Port 5 - Output data word 14 (INT bit14)
           TBEN_L4_8IOL:O.Data[80].15   // IO-Link Port 5 - Output data word 14 (INT bit15)
           TBEN_L4_8IOL:O.Data[80].2   // IO-Link Port 5 - Output data word 14 (INT bit2)
           TBEN_L4_8IOL:O.Data[80].3   // IO-Link Port 5 - Output data word 14 (INT bit3)
           TBEN_L4_8IOL:O.Data[80].4   // IO-Link Port 5 - Output data word 14 (INT bit4)
           TBEN_L4_8IOL:O.Data[80].5   // IO-Link Port 5 - Output data word 14 (INT bit5)
           TBEN_L4_8IOL:O.Data[80].6   // IO-Link Port 5 - Output data word 14 (INT bit6)
           TBEN_L4_8IOL:O.Data[80].7   // IO-Link Port 5 - Output data word 14 (INT bit7)
           TBEN_L4_8IOL:O.Data[80].8   // IO-Link Port 5 - Output data word 14 (INT bit8)
           TBEN_L4_8IOL:O.Data[80].9   // IO-Link Port 5 - Output data word 14 (INT bit9)
           TBEN_L4_8IOL:O.Data[81]   // IO-Link Port 5 - Output data word 15
           TBEN_L4_8IOL:O.Data[81].0   // IO-Link Port 5 - Output data word 15 (INT bit0)
           TBEN_L4_8IOL:O.Data[81].1   // IO-Link Port 5 - Output data word 15 (INT bit1)
           TBEN_L4_8IOL:O.Data[81].10   // IO-Link Port 5 - Output data word 15 (INT bit10)
           TBEN_L4_8IOL:O.Data[81].11   // IO-Link Port 5 - Output data word 15 (INT bit11)
           TBEN_L4_8IOL:O.Data[81].12   // IO-Link Port 5 - Output data word 15 (INT bit12)
           TBEN_L4_8IOL:O.Data[81].13   // IO-Link Port 5 - Output data word 15 (INT bit13)
           TBEN_L4_8IOL:O.Data[81].14   // IO-Link Port 5 - Output data word 15 (INT bit14)
           TBEN_L4_8IOL:O.Data[81].15   // IO-Link Port 5 - Output data word 15 (INT bit15)
           TBEN_L4_8IOL:O.Data[81].2   // IO-Link Port 5 - Output data word 15 (INT bit2)
           TBEN_L4_8IOL:O.Data[81].3   // IO-Link Port 5 - Output data word 15 (INT bit3)
           TBEN_L4_8IOL:O.Data[81].4   // IO-Link Port 5 - Output data word 15 (INT bit4)
           TBEN_L4_8IOL:O.Data[81].5   // IO-Link Port 5 - Output data word 15 (INT bit5)
           TBEN_L4_8IOL:O.Data[81].6   // IO-Link Port 5 - Output data word 15 (INT bit6)
           TBEN_L4_8IOL:O.Data[81].7   // IO-Link Port 5 - Output data word 15 (INT bit7)
           TBEN_L4_8IOL:O.Data[81].8   // IO-Link Port 5 - Output data word 15 (INT bit8)
           TBEN_L4_8IOL:O.Data[81].9   // IO-Link Port 5 - Output data word 15 (INT bit9)
           TBEN_L4_8IOL:O.Data[82]   // IO-Link Port 6 - Output data word 0
           TBEN_L4_8IOL:O.Data[82].0   // IO-Link Port 6 - Output data word 0 (INT bit0)
           TBEN_L4_8IOL:O.Data[82].1   // IO-Link Port 6 - Output data word 0 (INT bit1)
           TBEN_L4_8IOL:O.Data[82].10   // IO-Link Port 6 - Output data word 0 (INT bit10)
           TBEN_L4_8IOL:O.Data[82].11   // IO-Link Port 6 - Output data word 0 (INT bit11)
           TBEN_L4_8IOL:O.Data[82].12   // IO-Link Port 6 - Output data word 0 (INT bit12)
           TBEN_L4_8IOL:O.Data[82].13   // IO-Link Port 6 - Output data word 0 (INT bit13)
           TBEN_L4_8IOL:O.Data[82].14   // IO-Link Port 6 - Output data word 0 (INT bit14)
           TBEN_L4_8IOL:O.Data[82].15   // IO-Link Port 6 - Output data word 0 (INT bit15)
           TBEN_L4_8IOL:O.Data[82].2   // IO-Link Port 6 - Output data word 0 (INT bit2)
           TBEN_L4_8IOL:O.Data[82].3   // IO-Link Port 6 - Output data word 0 (INT bit3)
           TBEN_L4_8IOL:O.Data[82].4   // IO-Link Port 6 - Output data word 0 (INT bit4)
           TBEN_L4_8IOL:O.Data[82].5   // IO-Link Port 6 - Output data word 0 (INT bit5)
           TBEN_L4_8IOL:O.Data[82].6   // IO-Link Port 6 - Output data word 0 (INT bit6)
           TBEN_L4_8IOL:O.Data[82].7   // IO-Link Port 6 - Output data word 0 (INT bit7)
           TBEN_L4_8IOL:O.Data[82].8   // IO-Link Port 6 - Output data word 0 (INT bit8)
           TBEN_L4_8IOL:O.Data[82].9   // IO-Link Port 6 - Output data word 0 (INT bit9)
           TBEN_L4_8IOL:O.Data[83]   // IO-Link Port 6 - Output data word 1
           TBEN_L4_8IOL:O.Data[83].0   // IO-Link Port 6 - Output data word 1 (INT bit0)
           TBEN_L4_8IOL:O.Data[83].1   // IO-Link Port 6 - Output data word 1 (INT bit1)
           TBEN_L4_8IOL:O.Data[83].10   // IO-Link Port 6 - Output data word 1 (INT bit10)
           TBEN_L4_8IOL:O.Data[83].11   // IO-Link Port 6 - Output data word 1 (INT bit11)
           TBEN_L4_8IOL:O.Data[83].12   // IO-Link Port 6 - Output data word 1 (INT bit12)
           TBEN_L4_8IOL:O.Data[83].13   // IO-Link Port 6 - Output data word 1 (INT bit13)
           TBEN_L4_8IOL:O.Data[83].14   // IO-Link Port 6 - Output data word 1 (INT bit14)
           TBEN_L4_8IOL:O.Data[83].15   // IO-Link Port 6 - Output data word 1 (INT bit15)
           TBEN_L4_8IOL:O.Data[83].2   // IO-Link Port 6 - Output data word 1 (INT bit2)
           TBEN_L4_8IOL:O.Data[83].3   // IO-Link Port 6 - Output data word 1 (INT bit3)
           TBEN_L4_8IOL:O.Data[83].4   // IO-Link Port 6 - Output data word 1 (INT bit4)
           TBEN_L4_8IOL:O.Data[83].5   // IO-Link Port 6 - Output data word 1 (INT bit5)
           TBEN_L4_8IOL:O.Data[83].6   // IO-Link Port 6 - Output data word 1 (INT bit6)
           TBEN_L4_8IOL:O.Data[83].7   // IO-Link Port 6 - Output data word 1 (INT bit7)
           TBEN_L4_8IOL:O.Data[83].8   // IO-Link Port 6 - Output data word 1 (INT bit8)
           TBEN_L4_8IOL:O.Data[83].9   // IO-Link Port 6 - Output data word 1 (INT bit9)
           TBEN_L4_8IOL:O.Data[84]   // IO-Link Port 6 - Output data word 2
           TBEN_L4_8IOL:O.Data[84].0   // IO-Link Port 6 - Output data word 2 (INT bit0)
           TBEN_L4_8IOL:O.Data[84].1   // IO-Link Port 6 - Output data word 2 (INT bit1)
           TBEN_L4_8IOL:O.Data[84].10   // IO-Link Port 6 - Output data word 2 (INT bit10)
           TBEN_L4_8IOL:O.Data[84].11   // IO-Link Port 6 - Output data word 2 (INT bit11)
           TBEN_L4_8IOL:O.Data[84].12   // IO-Link Port 6 - Output data word 2 (INT bit12)
           TBEN_L4_8IOL:O.Data[84].13   // IO-Link Port 6 - Output data word 2 (INT bit13)
           TBEN_L4_8IOL:O.Data[84].14   // IO-Link Port 6 - Output data word 2 (INT bit14)
           TBEN_L4_8IOL:O.Data[84].15   // IO-Link Port 6 - Output data word 2 (INT bit15)
           TBEN_L4_8IOL:O.Data[84].2   // IO-Link Port 6 - Output data word 2 (INT bit2)
           TBEN_L4_8IOL:O.Data[84].3   // IO-Link Port 6 - Output data word 2 (INT bit3)
           TBEN_L4_8IOL:O.Data[84].4   // IO-Link Port 6 - Output data word 2 (INT bit4)
           TBEN_L4_8IOL:O.Data[84].5   // IO-Link Port 6 - Output data word 2 (INT bit5)
           TBEN_L4_8IOL:O.Data[84].6   // IO-Link Port 6 - Output data word 2 (INT bit6)
           TBEN_L4_8IOL:O.Data[84].7   // IO-Link Port 6 - Output data word 2 (INT bit7)
           TBEN_L4_8IOL:O.Data[84].8   // IO-Link Port 6 - Output data word 2 (INT bit8)
           TBEN_L4_8IOL:O.Data[84].9   // IO-Link Port 6 - Output data word 2 (INT bit9)
           TBEN_L4_8IOL:O.Data[85]   // IO-Link Port 6 - Output data word 3
           TBEN_L4_8IOL:O.Data[85].0   // IO-Link Port 6 - Output data word 3 (INT bit0)
           TBEN_L4_8IOL:O.Data[85].1   // IO-Link Port 6 - Output data word 3 (INT bit1)
           TBEN_L4_8IOL:O.Data[85].10   // IO-Link Port 6 - Output data word 3 (INT bit10)
           TBEN_L4_8IOL:O.Data[85].11   // IO-Link Port 6 - Output data word 3 (INT bit11)
           TBEN_L4_8IOL:O.Data[85].12   // IO-Link Port 6 - Output data word 3 (INT bit12)
           TBEN_L4_8IOL:O.Data[85].13   // IO-Link Port 6 - Output data word 3 (INT bit13)
           TBEN_L4_8IOL:O.Data[85].14   // IO-Link Port 6 - Output data word 3 (INT bit14)
           TBEN_L4_8IOL:O.Data[85].15   // IO-Link Port 6 - Output data word 3 (INT bit15)
           TBEN_L4_8IOL:O.Data[85].2   // IO-Link Port 6 - Output data word 3 (INT bit2)
           TBEN_L4_8IOL:O.Data[85].3   // IO-Link Port 6 - Output data word 3 (INT bit3)
           TBEN_L4_8IOL:O.Data[85].4   // IO-Link Port 6 - Output data word 3 (INT bit4)
           TBEN_L4_8IOL:O.Data[85].5   // IO-Link Port 6 - Output data word 3 (INT bit5)
           TBEN_L4_8IOL:O.Data[85].6   // IO-Link Port 6 - Output data word 3 (INT bit6)
           TBEN_L4_8IOL:O.Data[85].7   // IO-Link Port 6 - Output data word 3 (INT bit7)
           TBEN_L4_8IOL:O.Data[85].8   // IO-Link Port 6 - Output data word 3 (INT bit8)
           TBEN_L4_8IOL:O.Data[85].9   // IO-Link Port 6 - Output data word 3 (INT bit9)
           TBEN_L4_8IOL:O.Data[86]   // IO-Link Port 6 - Output data word 4
           TBEN_L4_8IOL:O.Data[86].0   // IO-Link Port 6 - Output data word 4 (INT bit0)
           TBEN_L4_8IOL:O.Data[86].1   // IO-Link Port 6 - Output data word 4 (INT bit1)
           TBEN_L4_8IOL:O.Data[86].10   // IO-Link Port 6 - Output data word 4 (INT bit10)
           TBEN_L4_8IOL:O.Data[86].11   // IO-Link Port 6 - Output data word 4 (INT bit11)
           TBEN_L4_8IOL:O.Data[86].12   // IO-Link Port 6 - Output data word 4 (INT bit12)
           TBEN_L4_8IOL:O.Data[86].13   // IO-Link Port 6 - Output data word 4 (INT bit13)
           TBEN_L4_8IOL:O.Data[86].14   // IO-Link Port 6 - Output data word 4 (INT bit14)
           TBEN_L4_8IOL:O.Data[86].15   // IO-Link Port 6 - Output data word 4 (INT bit15)
           TBEN_L4_8IOL:O.Data[86].2   // IO-Link Port 6 - Output data word 4 (INT bit2)
           TBEN_L4_8IOL:O.Data[86].3   // IO-Link Port 6 - Output data word 4 (INT bit3)
           TBEN_L4_8IOL:O.Data[86].4   // IO-Link Port 6 - Output data word 4 (INT bit4)
           TBEN_L4_8IOL:O.Data[86].5   // IO-Link Port 6 - Output data word 4 (INT bit5)
           TBEN_L4_8IOL:O.Data[86].6   // IO-Link Port 6 - Output data word 4 (INT bit6)
           TBEN_L4_8IOL:O.Data[86].7   // IO-Link Port 6 - Output data word 4 (INT bit7)
           TBEN_L4_8IOL:O.Data[86].8   // IO-Link Port 6 - Output data word 4 (INT bit8)
           TBEN_L4_8IOL:O.Data[86].9   // IO-Link Port 6 - Output data word 4 (INT bit9)
           TBEN_L4_8IOL:O.Data[87]   // IO-Link Port 6 - Output data word 5
           TBEN_L4_8IOL:O.Data[87].0   // IO-Link Port 6 - Output data word 5 (INT bit0)
           TBEN_L4_8IOL:O.Data[87].1   // IO-Link Port 6 - Output data word 5 (INT bit1)
           TBEN_L4_8IOL:O.Data[87].10   // IO-Link Port 6 - Output data word 5 (INT bit10)
           TBEN_L4_8IOL:O.Data[87].11   // IO-Link Port 6 - Output data word 5 (INT bit11)
           TBEN_L4_8IOL:O.Data[87].12   // IO-Link Port 6 - Output data word 5 (INT bit12)
           TBEN_L4_8IOL:O.Data[87].13   // IO-Link Port 6 - Output data word 5 (INT bit13)
           TBEN_L4_8IOL:O.Data[87].14   // IO-Link Port 6 - Output data word 5 (INT bit14)
           TBEN_L4_8IOL:O.Data[87].15   // IO-Link Port 6 - Output data word 5 (INT bit15)
           TBEN_L4_8IOL:O.Data[87].2   // IO-Link Port 6 - Output data word 5 (INT bit2)
           TBEN_L4_8IOL:O.Data[87].3   // IO-Link Port 6 - Output data word 5 (INT bit3)
           TBEN_L4_8IOL:O.Data[87].4   // IO-Link Port 6 - Output data word 5 (INT bit4)
           TBEN_L4_8IOL:O.Data[87].5   // IO-Link Port 6 - Output data word 5 (INT bit5)
           TBEN_L4_8IOL:O.Data[87].6   // IO-Link Port 6 - Output data word 5 (INT bit6)
           TBEN_L4_8IOL:O.Data[87].7   // IO-Link Port 6 - Output data word 5 (INT bit7)
           TBEN_L4_8IOL:O.Data[87].8   // IO-Link Port 6 - Output data word 5 (INT bit8)
           TBEN_L4_8IOL:O.Data[87].9   // IO-Link Port 6 - Output data word 5 (INT bit9)
           TBEN_L4_8IOL:O.Data[88]   // IO-Link Port 6 - Output data word 6
           TBEN_L4_8IOL:O.Data[88].0   // IO-Link Port 6 - Output data word 6 (INT bit0)
           TBEN_L4_8IOL:O.Data[88].1   // IO-Link Port 6 - Output data word 6 (INT bit1)
           TBEN_L4_8IOL:O.Data[88].10   // IO-Link Port 6 - Output data word 6 (INT bit10)
           TBEN_L4_8IOL:O.Data[88].11   // IO-Link Port 6 - Output data word 6 (INT bit11)
           TBEN_L4_8IOL:O.Data[88].12   // IO-Link Port 6 - Output data word 6 (INT bit12)
           TBEN_L4_8IOL:O.Data[88].13   // IO-Link Port 6 - Output data word 6 (INT bit13)
           TBEN_L4_8IOL:O.Data[88].14   // IO-Link Port 6 - Output data word 6 (INT bit14)
           TBEN_L4_8IOL:O.Data[88].15   // IO-Link Port 6 - Output data word 6 (INT bit15)
           TBEN_L4_8IOL:O.Data[88].2   // IO-Link Port 6 - Output data word 6 (INT bit2)
           TBEN_L4_8IOL:O.Data[88].3   // IO-Link Port 6 - Output data word 6 (INT bit3)
           TBEN_L4_8IOL:O.Data[88].4   // IO-Link Port 6 - Output data word 6 (INT bit4)
           TBEN_L4_8IOL:O.Data[88].5   // IO-Link Port 6 - Output data word 6 (INT bit5)
           TBEN_L4_8IOL:O.Data[88].6   // IO-Link Port 6 - Output data word 6 (INT bit6)
           TBEN_L4_8IOL:O.Data[88].7   // IO-Link Port 6 - Output data word 6 (INT bit7)
           TBEN_L4_8IOL:O.Data[88].8   // IO-Link Port 6 - Output data word 6 (INT bit8)
           TBEN_L4_8IOL:O.Data[88].9   // IO-Link Port 6 - Output data word 6 (INT bit9)
           TBEN_L4_8IOL:O.Data[89]   // IO-Link Port 6 - Output data word 7
           TBEN_L4_8IOL:O.Data[89].0   // IO-Link Port 6 - Output data word 7 (INT bit0)
           TBEN_L4_8IOL:O.Data[89].1   // IO-Link Port 6 - Output data word 7 (INT bit1)
           TBEN_L4_8IOL:O.Data[89].10   // IO-Link Port 6 - Output data word 7 (INT bit10)
           TBEN_L4_8IOL:O.Data[89].11   // IO-Link Port 6 - Output data word 7 (INT bit11)
           TBEN_L4_8IOL:O.Data[89].12   // IO-Link Port 6 - Output data word 7 (INT bit12)
           TBEN_L4_8IOL:O.Data[89].13   // IO-Link Port 6 - Output data word 7 (INT bit13)
           TBEN_L4_8IOL:O.Data[89].14   // IO-Link Port 6 - Output data word 7 (INT bit14)
           TBEN_L4_8IOL:O.Data[89].15   // IO-Link Port 6 - Output data word 7 (INT bit15)
           TBEN_L4_8IOL:O.Data[89].2   // IO-Link Port 6 - Output data word 7 (INT bit2)
           TBEN_L4_8IOL:O.Data[89].3   // IO-Link Port 6 - Output data word 7 (INT bit3)
           TBEN_L4_8IOL:O.Data[89].4   // IO-Link Port 6 - Output data word 7 (INT bit4)
           TBEN_L4_8IOL:O.Data[89].5   // IO-Link Port 6 - Output data word 7 (INT bit5)
           TBEN_L4_8IOL:O.Data[89].6   // IO-Link Port 6 - Output data word 7 (INT bit6)
           TBEN_L4_8IOL:O.Data[89].7   // IO-Link Port 6 - Output data word 7 (INT bit7)
           TBEN_L4_8IOL:O.Data[89].8   // IO-Link Port 6 - Output data word 7 (INT bit8)
           TBEN_L4_8IOL:O.Data[89].9   // IO-Link Port 6 - Output data word 7 (INT bit9)
           TBEN_L4_8IOL:O.Data[8]   // IO-Link Port 1 - Output data word 6
           TBEN_L4_8IOL:O.Data[8].0   // IO-Link Port 1 - Output data word 6 (INT bit0)
           TBEN_L4_8IOL:O.Data[8].1   // IO-Link Port 1 - Output data word 6 (INT bit1)
           TBEN_L4_8IOL:O.Data[8].10   // IO-Link Port 1 - Output data word 6 (INT bit10)
           TBEN_L4_8IOL:O.Data[8].11   // IO-Link Port 1 - Output data word 6 (INT bit11)
           TBEN_L4_8IOL:O.Data[8].12   // IO-Link Port 1 - Output data word 6 (INT bit12)
           TBEN_L4_8IOL:O.Data[8].13   // IO-Link Port 1 - Output data word 6 (INT bit13)
           TBEN_L4_8IOL:O.Data[8].14   // IO-Link Port 1 - Output data word 6 (INT bit14)
           TBEN_L4_8IOL:O.Data[8].15   // IO-Link Port 1 - Output data word 6 (INT bit15)
           TBEN_L4_8IOL:O.Data[8].2   // IO-Link Port 1 - Output data word 6 (INT bit2)
           TBEN_L4_8IOL:O.Data[8].3   // IO-Link Port 1 - Output data word 6 (INT bit3)
           TBEN_L4_8IOL:O.Data[8].4   // IO-Link Port 1 - Output data word 6 (INT bit4)
           TBEN_L4_8IOL:O.Data[8].5   // IO-Link Port 1 - Output data word 6 (INT bit5)
           TBEN_L4_8IOL:O.Data[8].6   // IO-Link Port 1 - Output data word 6 (INT bit6)
           TBEN_L4_8IOL:O.Data[8].7   // IO-Link Port 1 - Output data word 6 (INT bit7)
           TBEN_L4_8IOL:O.Data[8].8   // IO-Link Port 1 - Output data word 6 (INT bit8)
           TBEN_L4_8IOL:O.Data[8].9   // IO-Link Port 1 - Output data word 6 (INT bit9)
           TBEN_L4_8IOL:O.Data[90]   // IO-Link Port 6 - Output data word 8
           TBEN_L4_8IOL:O.Data[90].0   // IO-Link Port 6 - Output data word 8 (INT bit0)
           TBEN_L4_8IOL:O.Data[90].1   // IO-Link Port 6 - Output data word 8 (INT bit1)
           TBEN_L4_8IOL:O.Data[90].10   // IO-Link Port 6 - Output data word 8 (INT bit10)
           TBEN_L4_8IOL:O.Data[90].11   // IO-Link Port 6 - Output data word 8 (INT bit11)
           TBEN_L4_8IOL:O.Data[90].12   // IO-Link Port 6 - Output data word 8 (INT bit12)
           TBEN_L4_8IOL:O.Data[90].13   // IO-Link Port 6 - Output data word 8 (INT bit13)
           TBEN_L4_8IOL:O.Data[90].14   // IO-Link Port 6 - Output data word 8 (INT bit14)
           TBEN_L4_8IOL:O.Data[90].15   // IO-Link Port 6 - Output data word 8 (INT bit15)
           TBEN_L4_8IOL:O.Data[90].2   // IO-Link Port 6 - Output data word 8 (INT bit2)
           TBEN_L4_8IOL:O.Data[90].3   // IO-Link Port 6 - Output data word 8 (INT bit3)
           TBEN_L4_8IOL:O.Data[90].4   // IO-Link Port 6 - Output data word 8 (INT bit4)
           TBEN_L4_8IOL:O.Data[90].5   // IO-Link Port 6 - Output data word 8 (INT bit5)
           TBEN_L4_8IOL:O.Data[90].6   // IO-Link Port 6 - Output data word 8 (INT bit6)
           TBEN_L4_8IOL:O.Data[90].7   // IO-Link Port 6 - Output data word 8 (INT bit7)
           TBEN_L4_8IOL:O.Data[90].8   // IO-Link Port 6 - Output data word 8 (INT bit8)
           TBEN_L4_8IOL:O.Data[90].9   // IO-Link Port 6 - Output data word 8 (INT bit9)
           TBEN_L4_8IOL:O.Data[91]   // IO-Link Port 6 - Output data word 9
           TBEN_L4_8IOL:O.Data[91].0   // IO-Link Port 6 - Output data word 9 (INT bit0)
           TBEN_L4_8IOL:O.Data[91].1   // IO-Link Port 6 - Output data word 9 (INT bit1)
           TBEN_L4_8IOL:O.Data[91].10   // IO-Link Port 6 - Output data word 9 (INT bit10)
           TBEN_L4_8IOL:O.Data[91].11   // IO-Link Port 6 - Output data word 9 (INT bit11)
           TBEN_L4_8IOL:O.Data[91].12   // IO-Link Port 6 - Output data word 9 (INT bit12)
           TBEN_L4_8IOL:O.Data[91].13   // IO-Link Port 6 - Output data word 9 (INT bit13)
           TBEN_L4_8IOL:O.Data[91].14   // IO-Link Port 6 - Output data word 9 (INT bit14)
           TBEN_L4_8IOL:O.Data[91].15   // IO-Link Port 6 - Output data word 9 (INT bit15)
           TBEN_L4_8IOL:O.Data[91].2   // IO-Link Port 6 - Output data word 9 (INT bit2)
           TBEN_L4_8IOL:O.Data[91].3   // IO-Link Port 6 - Output data word 9 (INT bit3)
           TBEN_L4_8IOL:O.Data[91].4   // IO-Link Port 6 - Output data word 9 (INT bit4)
           TBEN_L4_8IOL:O.Data[91].5   // IO-Link Port 6 - Output data word 9 (INT bit5)
           TBEN_L4_8IOL:O.Data[91].6   // IO-Link Port 6 - Output data word 9 (INT bit6)
           TBEN_L4_8IOL:O.Data[91].7   // IO-Link Port 6 - Output data word 9 (INT bit7)
           TBEN_L4_8IOL:O.Data[91].8   // IO-Link Port 6 - Output data word 9 (INT bit8)
           TBEN_L4_8IOL:O.Data[91].9   // IO-Link Port 6 - Output data word 9 (INT bit9)
           TBEN_L4_8IOL:O.Data[92]   // IO-Link Port 6 - Output data word 10
           TBEN_L4_8IOL:O.Data[92].0   // IO-Link Port 6 - Output data word 10 (INT bit0)
           TBEN_L4_8IOL:O.Data[92].1   // IO-Link Port 6 - Output data word 10 (INT bit1)
           TBEN_L4_8IOL:O.Data[92].10   // IO-Link Port 6 - Output data word 10 (INT bit10)
           TBEN_L4_8IOL:O.Data[92].11   // IO-Link Port 6 - Output data word 10 (INT bit11)
           TBEN_L4_8IOL:O.Data[92].12   // IO-Link Port 6 - Output data word 10 (INT bit12)
           TBEN_L4_8IOL:O.Data[92].13   // IO-Link Port 6 - Output data word 10 (INT bit13)
           TBEN_L4_8IOL:O.Data[92].14   // IO-Link Port 6 - Output data word 10 (INT bit14)
           TBEN_L4_8IOL:O.Data[92].15   // IO-Link Port 6 - Output data word 10 (INT bit15)
           TBEN_L4_8IOL:O.Data[92].2   // IO-Link Port 6 - Output data word 10 (INT bit2)
           TBEN_L4_8IOL:O.Data[92].3   // IO-Link Port 6 - Output data word 10 (INT bit3)
           TBEN_L4_8IOL:O.Data[92].4   // IO-Link Port 6 - Output data word 10 (INT bit4)
           TBEN_L4_8IOL:O.Data[92].5   // IO-Link Port 6 - Output data word 10 (INT bit5)
           TBEN_L4_8IOL:O.Data[92].6   // IO-Link Port 6 - Output data word 10 (INT bit6)
           TBEN_L4_8IOL:O.Data[92].7   // IO-Link Port 6 - Output data word 10 (INT bit7)
           TBEN_L4_8IOL:O.Data[92].8   // IO-Link Port 6 - Output data word 10 (INT bit8)
           TBEN_L4_8IOL:O.Data[92].9   // IO-Link Port 6 - Output data word 10 (INT bit9)
           TBEN_L4_8IOL:O.Data[93]   // IO-Link Port 6 - Output data word 11
           TBEN_L4_8IOL:O.Data[93].0   // IO-Link Port 6 - Output data word 11 (INT bit0)
           TBEN_L4_8IOL:O.Data[93].1   // IO-Link Port 6 - Output data word 11 (INT bit1)
           TBEN_L4_8IOL:O.Data[93].10   // IO-Link Port 6 - Output data word 11 (INT bit10)
           TBEN_L4_8IOL:O.Data[93].11   // IO-Link Port 6 - Output data word 11 (INT bit11)
           TBEN_L4_8IOL:O.Data[93].12   // IO-Link Port 6 - Output data word 11 (INT bit12)
           TBEN_L4_8IOL:O.Data[93].13   // IO-Link Port 6 - Output data word 11 (INT bit13)
           TBEN_L4_8IOL:O.Data[93].14   // IO-Link Port 6 - Output data word 11 (INT bit14)
           TBEN_L4_8IOL:O.Data[93].15   // IO-Link Port 6 - Output data word 11 (INT bit15)
           TBEN_L4_8IOL:O.Data[93].2   // IO-Link Port 6 - Output data word 11 (INT bit2)
           TBEN_L4_8IOL:O.Data[93].3   // IO-Link Port 6 - Output data word 11 (INT bit3)
           TBEN_L4_8IOL:O.Data[93].4   // IO-Link Port 6 - Output data word 11 (INT bit4)
           TBEN_L4_8IOL:O.Data[93].5   // IO-Link Port 6 - Output data word 11 (INT bit5)
           TBEN_L4_8IOL:O.Data[93].6   // IO-Link Port 6 - Output data word 11 (INT bit6)
           TBEN_L4_8IOL:O.Data[93].7   // IO-Link Port 6 - Output data word 11 (INT bit7)
           TBEN_L4_8IOL:O.Data[93].8   // IO-Link Port 6 - Output data word 11 (INT bit8)
           TBEN_L4_8IOL:O.Data[93].9   // IO-Link Port 6 - Output data word 11 (INT bit9)
           TBEN_L4_8IOL:O.Data[94]   // IO-Link Port 6 - Output data word 12
           TBEN_L4_8IOL:O.Data[94].0   // IO-Link Port 6 - Output data word 12 (INT bit0)
           TBEN_L4_8IOL:O.Data[94].1   // IO-Link Port 6 - Output data word 12 (INT bit1)
           TBEN_L4_8IOL:O.Data[94].10   // IO-Link Port 6 - Output data word 12 (INT bit10)
           TBEN_L4_8IOL:O.Data[94].11   // IO-Link Port 6 - Output data word 12 (INT bit11)
           TBEN_L4_8IOL:O.Data[94].12   // IO-Link Port 6 - Output data word 12 (INT bit12)
           TBEN_L4_8IOL:O.Data[94].13   // IO-Link Port 6 - Output data word 12 (INT bit13)
           TBEN_L4_8IOL:O.Data[94].14   // IO-Link Port 6 - Output data word 12 (INT bit14)
           TBEN_L4_8IOL:O.Data[94].15   // IO-Link Port 6 - Output data word 12 (INT bit15)
           TBEN_L4_8IOL:O.Data[94].2   // IO-Link Port 6 - Output data word 12 (INT bit2)
           TBEN_L4_8IOL:O.Data[94].3   // IO-Link Port 6 - Output data word 12 (INT bit3)
           TBEN_L4_8IOL:O.Data[94].4   // IO-Link Port 6 - Output data word 12 (INT bit4)
           TBEN_L4_8IOL:O.Data[94].5   // IO-Link Port 6 - Output data word 12 (INT bit5)
           TBEN_L4_8IOL:O.Data[94].6   // IO-Link Port 6 - Output data word 12 (INT bit6)
           TBEN_L4_8IOL:O.Data[94].7   // IO-Link Port 6 - Output data word 12 (INT bit7)
           TBEN_L4_8IOL:O.Data[94].8   // IO-Link Port 6 - Output data word 12 (INT bit8)
           TBEN_L4_8IOL:O.Data[94].9   // IO-Link Port 6 - Output data word 12 (INT bit9)
           TBEN_L4_8IOL:O.Data[95]   // IO-Link Port 6 - Output data word 13
           TBEN_L4_8IOL:O.Data[95].0   // IO-Link Port 6 - Output data word 13 (INT bit0)
           TBEN_L4_8IOL:O.Data[95].1   // IO-Link Port 6 - Output data word 13 (INT bit1)
           TBEN_L4_8IOL:O.Data[95].10   // IO-Link Port 6 - Output data word 13 (INT bit10)
           TBEN_L4_8IOL:O.Data[95].11   // IO-Link Port 6 - Output data word 13 (INT bit11)
           TBEN_L4_8IOL:O.Data[95].12   // IO-Link Port 6 - Output data word 13 (INT bit12)
           TBEN_L4_8IOL:O.Data[95].13   // IO-Link Port 6 - Output data word 13 (INT bit13)
           TBEN_L4_8IOL:O.Data[95].14   // IO-Link Port 6 - Output data word 13 (INT bit14)
           TBEN_L4_8IOL:O.Data[95].15   // IO-Link Port 6 - Output data word 13 (INT bit15)
           TBEN_L4_8IOL:O.Data[95].2   // IO-Link Port 6 - Output data word 13 (INT bit2)
           TBEN_L4_8IOL:O.Data[95].3   // IO-Link Port 6 - Output data word 13 (INT bit3)
           TBEN_L4_8IOL:O.Data[95].4   // IO-Link Port 6 - Output data word 13 (INT bit4)
           TBEN_L4_8IOL:O.Data[95].5   // IO-Link Port 6 - Output data word 13 (INT bit5)
           TBEN_L4_8IOL:O.Data[95].6   // IO-Link Port 6 - Output data word 13 (INT bit6)
           TBEN_L4_8IOL:O.Data[95].7   // IO-Link Port 6 - Output data word 13 (INT bit7)
           TBEN_L4_8IOL:O.Data[95].8   // IO-Link Port 6 - Output data word 13 (INT bit8)
           TBEN_L4_8IOL:O.Data[95].9   // IO-Link Port 6 - Output data word 13 (INT bit9)
           TBEN_L4_8IOL:O.Data[96]   // IO-Link Port 6 - Output data word 14
           TBEN_L4_8IOL:O.Data[96].0   // IO-Link Port 6 - Output data word 14 (INT bit0)
           TBEN_L4_8IOL:O.Data[96].1   // IO-Link Port 6 - Output data word 14 (INT bit1)
           TBEN_L4_8IOL:O.Data[96].10   // IO-Link Port 6 - Output data word 14 (INT bit10)
           TBEN_L4_8IOL:O.Data[96].11   // IO-Link Port 6 - Output data word 14 (INT bit11)
           TBEN_L4_8IOL:O.Data[96].12   // IO-Link Port 6 - Output data word 14 (INT bit12)
           TBEN_L4_8IOL:O.Data[96].13   // IO-Link Port 6 - Output data word 14 (INT bit13)
           TBEN_L4_8IOL:O.Data[96].14   // IO-Link Port 6 - Output data word 14 (INT bit14)
           TBEN_L4_8IOL:O.Data[96].15   // IO-Link Port 6 - Output data word 14 (INT bit15)
           TBEN_L4_8IOL:O.Data[96].2   // IO-Link Port 6 - Output data word 14 (INT bit2)
           TBEN_L4_8IOL:O.Data[96].3   // IO-Link Port 6 - Output data word 14 (INT bit3)
           TBEN_L4_8IOL:O.Data[96].4   // IO-Link Port 6 - Output data word 14 (INT bit4)
           TBEN_L4_8IOL:O.Data[96].5   // IO-Link Port 6 - Output data word 14 (INT bit5)
           TBEN_L4_8IOL:O.Data[96].6   // IO-Link Port 6 - Output data word 14 (INT bit6)
           TBEN_L4_8IOL:O.Data[96].7   // IO-Link Port 6 - Output data word 14 (INT bit7)
           TBEN_L4_8IOL:O.Data[96].8   // IO-Link Port 6 - Output data word 14 (INT bit8)
           TBEN_L4_8IOL:O.Data[96].9   // IO-Link Port 6 - Output data word 14 (INT bit9)
           TBEN_L4_8IOL:O.Data[97]   // IO-Link Port 6 - Output data word 15
           TBEN_L4_8IOL:O.Data[97].0   // IO-Link Port 6 - Output data word 15 (INT bit0)
           TBEN_L4_8IOL:O.Data[97].1   // IO-Link Port 6 - Output data word 15 (INT bit1)
           TBEN_L4_8IOL:O.Data[97].10   // IO-Link Port 6 - Output data word 15 (INT bit10)
           TBEN_L4_8IOL:O.Data[97].11   // IO-Link Port 6 - Output data word 15 (INT bit11)
           TBEN_L4_8IOL:O.Data[97].12   // IO-Link Port 6 - Output data word 15 (INT bit12)
           TBEN_L4_8IOL:O.Data[97].13   // IO-Link Port 6 - Output data word 15 (INT bit13)
           TBEN_L4_8IOL:O.Data[97].14   // IO-Link Port 6 - Output data word 15 (INT bit14)
           TBEN_L4_8IOL:O.Data[97].15   // IO-Link Port 6 - Output data word 15 (INT bit15)
           TBEN_L4_8IOL:O.Data[97].2   // IO-Link Port 6 - Output data word 15 (INT bit2)
           TBEN_L4_8IOL:O.Data[97].3   // IO-Link Port 6 - Output data word 15 (INT bit3)
           TBEN_L4_8IOL:O.Data[97].4   // IO-Link Port 6 - Output data word 15 (INT bit4)
           TBEN_L4_8IOL:O.Data[97].5   // IO-Link Port 6 - Output data word 15 (INT bit5)
           TBEN_L4_8IOL:O.Data[97].6   // IO-Link Port 6 - Output data word 15 (INT bit6)
           TBEN_L4_8IOL:O.Data[97].7   // IO-Link Port 6 - Output data word 15 (INT bit7)
           TBEN_L4_8IOL:O.Data[97].8   // IO-Link Port 6 - Output data word 15 (INT bit8)
           TBEN_L4_8IOL:O.Data[97].9   // IO-Link Port 6 - Output data word 15 (INT bit9)
           TBEN_L4_8IOL:O.Data[98]   // IO-Link Port 7 - Output data word 0
           TBEN_L4_8IOL:O.Data[98].0   // IO-Link Port 7 - Output data word 0 (INT bit0)
           TBEN_L4_8IOL:O.Data[98].1   // IO-Link Port 7 - Output data word 0 (INT bit1)
           TBEN_L4_8IOL:O.Data[98].10   // IO-Link Port 7 - Output data word 0 (INT bit10)
           TBEN_L4_8IOL:O.Data[98].11   // IO-Link Port 7 - Output data word 0 (INT bit11)
           TBEN_L4_8IOL:O.Data[98].12   // IO-Link Port 7 - Output data word 0 (INT bit12)
           TBEN_L4_8IOL:O.Data[98].13   // IO-Link Port 7 - Output data word 0 (INT bit13)
           TBEN_L4_8IOL:O.Data[98].14   // IO-Link Port 7 - Output data word 0 (INT bit14)
           TBEN_L4_8IOL:O.Data[98].15   // IO-Link Port 7 - Output data word 0 (INT bit15)
           TBEN_L4_8IOL:O.Data[98].2   // IO-Link Port 7 - Output data word 0 (INT bit2)
           TBEN_L4_8IOL:O.Data[98].3   // IO-Link Port 7 - Output data word 0 (INT bit3)
           TBEN_L4_8IOL:O.Data[98].4   // IO-Link Port 7 - Output data word 0 (INT bit4)
           TBEN_L4_8IOL:O.Data[98].5   // IO-Link Port 7 - Output data word 0 (INT bit5)
           TBEN_L4_8IOL:O.Data[98].6   // IO-Link Port 7 - Output data word 0 (INT bit6)
           TBEN_L4_8IOL:O.Data[98].7   // IO-Link Port 7 - Output data word 0 (INT bit7)
           TBEN_L4_8IOL:O.Data[98].8   // IO-Link Port 7 - Output data word 0 (INT bit8)
           TBEN_L4_8IOL:O.Data[98].9   // IO-Link Port 7 - Output data word 0 (INT bit9)
           TBEN_L4_8IOL:O.Data[99]   // IO-Link Port 7 - Output data word 1
           TBEN_L4_8IOL:O.Data[99].0   // IO-Link Port 7 - Output data word 1 (INT bit0)
           TBEN_L4_8IOL:O.Data[99].1   // IO-Link Port 7 - Output data word 1 (INT bit1)
           TBEN_L4_8IOL:O.Data[99].10   // IO-Link Port 7 - Output data word 1 (INT bit10)
           TBEN_L4_8IOL:O.Data[99].11   // IO-Link Port 7 - Output data word 1 (INT bit11)
           TBEN_L4_8IOL:O.Data[99].12   // IO-Link Port 7 - Output data word 1 (INT bit12)
           TBEN_L4_8IOL:O.Data[99].13   // IO-Link Port 7 - Output data word 1 (INT bit13)
           TBEN_L4_8IOL:O.Data[99].14   // IO-Link Port 7 - Output data word 1 (INT bit14)
           TBEN_L4_8IOL:O.Data[99].15   // IO-Link Port 7 - Output data word 1 (INT bit15)
           TBEN_L4_8IOL:O.Data[99].2   // IO-Link Port 7 - Output data word 1 (INT bit2)
           TBEN_L4_8IOL:O.Data[99].3   // IO-Link Port 7 - Output data word 1 (INT bit3)
           TBEN_L4_8IOL:O.Data[99].4   // IO-Link Port 7 - Output data word 1 (INT bit4)
           TBEN_L4_8IOL:O.Data[99].5   // IO-Link Port 7 - Output data word 1 (INT bit5)
           TBEN_L4_8IOL:O.Data[99].6   // IO-Link Port 7 - Output data word 1 (INT bit6)
           TBEN_L4_8IOL:O.Data[99].7   // IO-Link Port 7 - Output data word 1 (INT bit7)
           TBEN_L4_8IOL:O.Data[99].8   // IO-Link Port 7 - Output data word 1 (INT bit8)
           TBEN_L4_8IOL:O.Data[99].9   // IO-Link Port 7 - Output data word 1 (INT bit9)
           TBEN_L4_8IOL:O.Data[9]   // IO-Link Port 1 - Output data word 7
           TBEN_L4_8IOL:O.Data[9].0   // IO-Link Port 1 - Output data word 7 (INT bit0)
           TBEN_L4_8IOL:O.Data[9].1   // IO-Link Port 1 - Output data word 7 (INT bit1)
           TBEN_L4_8IOL:O.Data[9].10   // IO-Link Port 1 - Output data word 7 (INT bit10)
           TBEN_L4_8IOL:O.Data[9].11   // IO-Link Port 1 - Output data word 7 (INT bit11)
           TBEN_L4_8IOL:O.Data[9].12   // IO-Link Port 1 - Output data word 7 (INT bit12)
           TBEN_L4_8IOL:O.Data[9].13   // IO-Link Port 1 - Output data word 7 (INT bit13)
           TBEN_L4_8IOL:O.Data[9].14   // IO-Link Port 1 - Output data word 7 (INT bit14)
           TBEN_L4_8IOL:O.Data[9].15   // IO-Link Port 1 - Output data word 7 (INT bit15)
           TBEN_L4_8IOL:O.Data[9].2   // IO-Link Port 1 - Output data word 7 (INT bit2)
           TBEN_L4_8IOL:O.Data[9].3   // IO-Link Port 1 - Output data word 7 (INT bit3)
           TBEN_L4_8IOL:O.Data[9].4   // IO-Link Port 1 - Output data word 7 (INT bit4)
           TBEN_L4_8IOL:O.Data[9].5   // IO-Link Port 1 - Output data word 7 (INT bit5)
           TBEN_L4_8IOL:O.Data[9].6   // IO-Link Port 1 - Output data word 7 (INT bit6)
           TBEN_L4_8IOL:O.Data[9].7   // IO-Link Port 1 - Output data word 7 (INT bit7)
           TBEN_L4_8IOL:O.Data[9].8   // IO-Link Port 1 - Output data word 7 (INT bit8)
           TBEN_L4_8IOL:O.Data[9].9   // IO-Link Port 1 - Output data word 7 (INT bit9)
           TBEN_L4_8IOL:C.Data[100]   // IO-Link Port 6 - Cycle time
           TBEN_L4_8IOL:C.Data[0]   // Reserved
           TBEN_L4_8IOL:C.Data[101]   // IO-Link Port 6 - Revision
           TBEN_L4_8IOL:C.Data[100].0   // IO-Link Port 6 - Cycle time (ENUM bit0): 00000000=automatic, 00010000=1.6 ms, 00011000=2.4 ms, 00100000=3.2 ms, 00101000=4.0 ms, 00110000=4.8 ms, 00111000=5.6 ms, 01000000=6.4 ms, 01000010=7.2 ms, 01000100=8.0 ms, 01000110=8.8 ms, 01001000=9.6 ms
           TBEN_L4_8IOL:C.Data[100].1   // IO-Link Port 6 - Cycle time (ENUM bit1): 01001010=10.4 ms, 01001100=11.2 ms, 01001110=12.0 ms, 01010000=12.8 ms, 01010100=14.4 ms, 01011000=16.0 ms, 01011100=17.6 ms, 01100000=19.2 ms, 01100100=20.8 ms, 01101000=22.4 ms, 01101100=24.0 ms, 01110000=25.6 ms
           TBEN_L4_8IOL:C.Data[100].2   // IO-Link Port 6 - Cycle time (ENUM bit2): 01110100=27.2 ms, 01111000=28.8 ms, 01111100=30.4 ms, 10000000=32.0 ms, 10000001=33.6 ms, 10000010=35.2 ms, 10000011=36.8 ms, 10000100=38.4 ms, 10000101=40.0 ms, 10000110=41.6 ms, 10000111=43.2 ms, 10001000=44.8 ms
           TBEN_L4_8IOL:C.Data[100].3   // IO-Link Port 6 - Cycle time (ENUM bit3): 10001001=46.4 ms, 10001010=48.0 ms, 10001011=49.6 ms, 10001100=51.2 ms, 10001101=52.8 ms, 10001110=54.4 ms, 10001111=56.0 ms, 10010000=57.6 ms, 10010001=59.2 ms, 10010010=60.8 ms, 10010011=62.4 ms, 10010100=64.0 ms
           TBEN_L4_8IOL:C.Data[100].4   // IO-Link Port 6 - Cycle time (ENUM bit4): 10010101=65.6 ms, 10010110=67.2 ms, 10010111=68.8 ms, 10011000=70.4 ms, 10011001=72.0 ms, 10011010=73.6 ms, 10011011=75.2 ms, 10011100=76.8 ms, 10011101=78.4 ms, 10011110=80.0 ms, 10011111=81.6 ms
           TBEN_L4_8IOL:C.Data[100].5   // IO-Link Port 6 - Cycle time (ENUM bit5): 10100000=83.2 ms, 10100001=84.8 ms, 10100010=86.4 ms, 10100011=88.0 ms, 10100100=89.6 ms, 10100101=91.2 ms, 10100110=92.8 ms, 10100111=94.4 ms, 10101000=96.0 ms, 10101001=97.6 ms, 10101010=99.2 ms
           TBEN_L4_8IOL:C.Data[100].6   // IO-Link Port 6 - Cycle time (ENUM bit6): 10101011=100.8 ms, 10101100=102.4 ms, 10101101=104.0 ms, 10101110=105.6 ms, 10101111=107.2 ms, 10110000=108.8 ms, 10110001=110.4 ms, 10110010=112.0 ms, 10110011=113.6 ms, 10110100=115.2 ms, 10110101=116.8 ms
           TBEN_L4_8IOL:C.Data[100].7   // IO-Link Port 6 - Cycle time (ENUM bit7): 10110110=118.4 ms, 10110111=120.0 ms, 10111000=121.6 ms, 10111001=123.2 ms, 10111010=124.8 ms, 10111011=126.4 ms, 10111100=128.0 ms, 10111101=129.6 ms, 10111110=131.2 ms, 10111111=132.8 ms, 11111111=automatic, compatible
           TBEN_L4_8IOL:C.Data[101].0   // IO-Link Port 6 - Revision (ENUM bit0): 0=automatic, 1=V1.0
           TBEN_L4_8IOL:C.Data[101].1   // Reserved
           TBEN_L4_8IOL:C.Data[101].2   // Reserved
           TBEN_L4_8IOL:C.Data[101].3   // Reserved
           TBEN_L4_8IOL:C.Data[101].4   // Reserved
           TBEN_L4_8IOL:C.Data[101].5   // Reserved
           TBEN_L4_8IOL:C.Data[101].6   // Reserved
           TBEN_L4_8IOL:C.Data[101].7   // Reserved
           TBEN_L4_8IOL:C.Data[102]   // IO-Link Port 6 - Activate Quick Start-Up
           TBEN_L4_8IOL:C.Data[102].0   // IO-Link Port 6 - Activate Quick Start-Up (ENUM bit0): 0=no, 1=yes
           TBEN_L4_8IOL:C.Data[102].1   // Reserved
           TBEN_L4_8IOL:C.Data[102].2   // Reserved
           TBEN_L4_8IOL:C.Data[102].3   // Reserved
           TBEN_L4_8IOL:C.Data[102].4   // Reserved
           TBEN_L4_8IOL:C.Data[102].5   // Reserved
           TBEN_L4_8IOL:C.Data[102].6   // Reserved
           TBEN_L4_8IOL:C.Data[102].7   // Reserved
           TBEN_L4_8IOL:C.Data[103]   // IO-Link Port 6 - Device parametrization via GSD
           TBEN_L4_8IOL:C.Data[103].0   // IO-Link Port 6 - Device parametrization via GSD (ENUM bit0): 0=inactive, 1=active
           TBEN_L4_8IOL:C.Data[103].1   // Reserved
           TBEN_L4_8IOL:C.Data[103].2   // Reserved
           TBEN_L4_8IOL:C.Data[103].3   // Reserved
           TBEN_L4_8IOL:C.Data[103].4   // Reserved
           TBEN_L4_8IOL:C.Data[103].5   // Reserved
           TBEN_L4_8IOL:C.Data[103].6   // Reserved
           TBEN_L4_8IOL:C.Data[103].7   // Reserved
           TBEN_L4_8IOL:C.Data[104]   // IO-Link Port 6 - Process input data invalid
           TBEN_L4_8IOL:C.Data[104].0   // IO-Link Port 6 - Process input data invalid (ENUM bit0): 0=diagnostic generated, 1=no diagnostic generated
           TBEN_L4_8IOL:C.Data[104].1   // Reserved
           TBEN_L4_8IOL:C.Data[104].2   // Reserved
           TBEN_L4_8IOL:C.Data[104].3   // Reserved
           TBEN_L4_8IOL:C.Data[104].4   // Reserved
           TBEN_L4_8IOL:C.Data[104].5   // Reserved
           TBEN_L4_8IOL:C.Data[104].6   // Reserved
           TBEN_L4_8IOL:C.Data[104].7   // Reserved
           TBEN_L4_8IOL:C.Data[105]   // IO-Link Port 6 - Deactivate diagnostics
           TBEN_L4_8IOL:C.Data[105].0   // IO-Link Port 6 - Deactivate diagnostics (ENUM bit0): 00=no, 01=notifications
           TBEN_L4_8IOL:C.Data[105].1   // IO-Link Port 6 - Deactivate diagnostics (ENUM bit1): 10=notifications and warnings, 11=yes
           TBEN_L4_8IOL:C.Data[105].2   // Reserved
           TBEN_L4_8IOL:C.Data[105].3   // Reserved
           TBEN_L4_8IOL:C.Data[105].4   // Reserved
           TBEN_L4_8IOL:C.Data[105].5   // Reserved
           TBEN_L4_8IOL:C.Data[105].6   // Reserved
           TBEN_L4_8IOL:C.Data[105].7   // Reserved
           TBEN_L4_8IOL:C.Data[106]   // IO-Link Port 6 - Input data mapping
           TBEN_L4_8IOL:C.Data[106].0   // IO-Link Port 6 - Input data mapping (ENUM bit0): 00=direct, 01=swap 16 bit
           TBEN_L4_8IOL:C.Data[106].1   // IO-Link Port 6 - Input data mapping (ENUM bit1): 10=swap 32 bit, 11=swap
           TBEN_L4_8IOL:C.Data[106].2   // Reserved
           TBEN_L4_8IOL:C.Data[106].3   // Reserved
           TBEN_L4_8IOL:C.Data[106].4   // Reserved
           TBEN_L4_8IOL:C.Data[106].5   // Reserved
           TBEN_L4_8IOL:C.Data[106].6   // Reserved
           TBEN_L4_8IOL:C.Data[106].7   // Reserved
           TBEN_L4_8IOL:C.Data[107]   // IO-Link Port 6 - Output data mapping
           TBEN_L4_8IOL:C.Data[107].0   // IO-Link Port 6 - Output data mapping (ENUM bit0): 00=direct, 01=swap 16 bit
           TBEN_L4_8IOL:C.Data[107].1   // IO-Link Port 6 - Output data mapping (ENUM bit1): 10=swap 32 bit, 11=swap
           TBEN_L4_8IOL:C.Data[107].2   // Reserved
           TBEN_L4_8IOL:C.Data[107].3   // Reserved
           TBEN_L4_8IOL:C.Data[107].4   // Reserved
           TBEN_L4_8IOL:C.Data[107].5   // Reserved
           TBEN_L4_8IOL:C.Data[107].6   // Reserved
           TBEN_L4_8IOL:C.Data[107].7   // Reserved
           TBEN_L4_8IOL:C.Data[108]   // IO-Link Port 6 - Vendor ID
           TBEN_L4_8IOL:C.Data[108].0   // IO-Link Port 6 - Vendor ID (INT bit0)
           TBEN_L4_8IOL:C.Data[108].1   // IO-Link Port 6 - Vendor ID (INT bit1)
           TBEN_L4_8IOL:C.Data[108].2   // IO-Link Port 6 - Vendor ID (INT bit2)
           TBEN_L4_8IOL:C.Data[108].3   // IO-Link Port 6 - Vendor ID (INT bit3)
           TBEN_L4_8IOL:C.Data[108].4   // IO-Link Port 6 - Vendor ID (INT bit4)
           TBEN_L4_8IOL:C.Data[108].5   // IO-Link Port 6 - Vendor ID (INT bit5)
           TBEN_L4_8IOL:C.Data[108].6   // IO-Link Port 6 - Vendor ID (INT bit6)
           TBEN_L4_8IOL:C.Data[108].7   // IO-Link Port 6 - Vendor ID (INT bit7)
           TBEN_L4_8IOL:C.Data[109]   // IO-Link Port 6 - Vendor ID
           TBEN_L4_8IOL:C.Data[109].0   // IO-Link Port 6 - Vendor ID (INT bit8)
           TBEN_L4_8IOL:C.Data[109].1   // IO-Link Port 6 - Vendor ID (INT bit9)
           TBEN_L4_8IOL:C.Data[109].2   // IO-Link Port 6 - Vendor ID (INT bit10)
           TBEN_L4_8IOL:C.Data[109].3   // IO-Link Port 6 - Vendor ID (INT bit11)
           TBEN_L4_8IOL:C.Data[109].4   // IO-Link Port 6 - Vendor ID (INT bit12)
           TBEN_L4_8IOL:C.Data[109].5   // IO-Link Port 6 - Vendor ID (INT bit13)
           TBEN_L4_8IOL:C.Data[109].6   // IO-Link Port 6 - Vendor ID (INT bit14)
           TBEN_L4_8IOL:C.Data[109].7   // IO-Link Port 6 - Vendor ID (INT bit15)
           TBEN_L4_8IOL:C.Data[10]   // DXP 1 - Manual reset after overcurr.
           TBEN_L4_8IOL:C.Data[10].0   // DXP 1 - Manual reset after overcurr. (ENUM bit0): 0=no, 1=yes
           TBEN_L4_8IOL:C.Data[10].1   // Reserved
           TBEN_L4_8IOL:C.Data[10].2   // Reserved
           TBEN_L4_8IOL:C.Data[10].3   // Reserved
           TBEN_L4_8IOL:C.Data[10].4   // Reserved
           TBEN_L4_8IOL:C.Data[10].5   // Reserved
           TBEN_L4_8IOL:C.Data[10].6   // Reserved
           TBEN_L4_8IOL:C.Data[10].7   // Reserved
           TBEN_L4_8IOL:C.Data[110]   // IO-Link Port 6 - Device ID
           TBEN_L4_8IOL:C.Data[110].0   // IO-Link Port 6 - Device ID (INT bit0)
           TBEN_L4_8IOL:C.Data[110].1   // IO-Link Port 6 - Device ID (INT bit1)
           TBEN_L4_8IOL:C.Data[110].2   // IO-Link Port 6 - Device ID (INT bit2)
           TBEN_L4_8IOL:C.Data[110].3   // IO-Link Port 6 - Device ID (INT bit3)
           TBEN_L4_8IOL:C.Data[110].4   // IO-Link Port 6 - Device ID (INT bit4)
           TBEN_L4_8IOL:C.Data[110].5   // IO-Link Port 6 - Device ID (INT bit5)
           TBEN_L4_8IOL:C.Data[110].6   // IO-Link Port 6 - Device ID (INT bit6)
           TBEN_L4_8IOL:C.Data[110].7   // IO-Link Port 6 - Device ID (INT bit7)
           TBEN_L4_8IOL:C.Data[111]   // IO-Link Port 6 - Device ID
           TBEN_L4_8IOL:C.Data[111].0   // IO-Link Port 6 - Device ID (INT bit8)
           TBEN_L4_8IOL:C.Data[111].1   // IO-Link Port 6 - Device ID (INT bit9)
           TBEN_L4_8IOL:C.Data[111].2   // IO-Link Port 6 - Device ID (INT bit10)
           TBEN_L4_8IOL:C.Data[111].3   // IO-Link Port 6 - Device ID (INT bit11)
           TBEN_L4_8IOL:C.Data[111].4   // IO-Link Port 6 - Device ID (INT bit12)
           TBEN_L4_8IOL:C.Data[111].5   // IO-Link Port 6 - Device ID (INT bit13)
           TBEN_L4_8IOL:C.Data[111].6   // IO-Link Port 6 - Device ID (INT bit14)
           TBEN_L4_8IOL:C.Data[111].7   // IO-Link Port 6 - Device ID (INT bit15)
           TBEN_L4_8IOL:C.Data[112]   // IO-Link Port 6 - Device ID
           TBEN_L4_8IOL:C.Data[112].0   // IO-Link Port 6 - Device ID (INT bit16)
           TBEN_L4_8IOL:C.Data[112].1   // IO-Link Port 6 - Device ID (INT bit17)
           TBEN_L4_8IOL:C.Data[112].2   // IO-Link Port 6 - Device ID (INT bit18)
           TBEN_L4_8IOL:C.Data[112].3   // IO-Link Port 6 - Device ID (INT bit19)
           TBEN_L4_8IOL:C.Data[112].4   // IO-Link Port 6 - Device ID (INT bit20)
           TBEN_L4_8IOL:C.Data[112].5   // IO-Link Port 6 - Device ID (INT bit21)
           TBEN_L4_8IOL:C.Data[112].6   // IO-Link Port 6 - Device ID (INT bit22)
           TBEN_L4_8IOL:C.Data[112].7   // IO-Link Port 6 - Device ID (INT bit23)
           TBEN_L4_8IOL:C.Data[113]   // IO-Link Port 6 - Device ID
           TBEN_L4_8IOL:C.Data[113].0   // IO-Link Port 6 - Device ID (INT bit24)
           TBEN_L4_8IOL:C.Data[113].1   // IO-Link Port 6 - Device ID (INT bit25)
           TBEN_L4_8IOL:C.Data[113].2   // IO-Link Port 6 - Device ID (INT bit26)
           TBEN_L4_8IOL:C.Data[113].3   // IO-Link Port 6 - Device ID (INT bit27)
           TBEN_L4_8IOL:C.Data[113].4   // IO-Link Port 6 - Device ID (INT bit28)
           TBEN_L4_8IOL:C.Data[113].5   // IO-Link Port 6 - Device ID (INT bit29)
           TBEN_L4_8IOL:C.Data[113].6   // IO-Link Port 6 - Device ID (INT bit30)
           TBEN_L4_8IOL:C.Data[113].7   // IO-Link Port 6 - Device ID (INT bit31)
           TBEN_L4_8IOL:C.Data[114]   // IO-Link Port 7 - Operation mode
           TBEN_L4_8IOL:C.Data[114].0   // IO-Link Port 7 - Operation mode (ENUM bit0): 0000=IO-Link without validation, 0001=IO-Link with family compatible device
           TBEN_L4_8IOL:C.Data[114].1   // IO-Link Port 7 - Operation mode (ENUM bit1): 0010=IO-Link with compatible device, 0011=IO-Link with identical device
           TBEN_L4_8IOL:C.Data[114].2   // IO-Link Port 7 - Operation mode (ENUM bit2): 0100=DI (with parameter access)
           TBEN_L4_8IOL:C.Data[114].3   // IO-Link Port 7 - Operation mode (ENUM bit3): 1000=DI
           TBEN_L4_8IOL:C.Data[114].4   // Reserved
           TBEN_L4_8IOL:C.Data[114].5   // Reserved
           TBEN_L4_8IOL:C.Data[114].6   // Reserved
           TBEN_L4_8IOL:C.Data[114].7   // Reserved
           TBEN_L4_8IOL:C.Data[115]   // IO-Link Port 7 - Data storage mode
           TBEN_L4_8IOL:C.Data[115].0   // IO-Link Port 7 - Data storage mode (ENUM bit0): 00=activated, 01=overwrite
           TBEN_L4_8IOL:C.Data[115].1   // IO-Link Port 7 - Data storage mode (ENUM bit1): 10=read in, 11=deactivated, clear
           TBEN_L4_8IOL:C.Data[115].2   // Reserved
           TBEN_L4_8IOL:C.Data[115].3   // Reserved
           TBEN_L4_8IOL:C.Data[115].4   // Reserved
           TBEN_L4_8IOL:C.Data[115].5   // Reserved
           TBEN_L4_8IOL:C.Data[115].6   // Reserved
           TBEN_L4_8IOL:C.Data[115].7   // Reserved
           TBEN_L4_8IOL:C.Data[116]   // IO-Link Port 7 - Cycle time
           TBEN_L4_8IOL:C.Data[116].0   // IO-Link Port 7 - Cycle time (ENUM bit0): 00000000=automatic, 00010000=1.6 ms, 00011000=2.4 ms, 00100000=3.2 ms, 00101000=4.0 ms, 00110000=4.8 ms, 00111000=5.6 ms, 01000000=6.4 ms, 01000010=7.2 ms, 01000100=8.0 ms, 01000110=8.8 ms, 01001000=9.6 ms
           TBEN_L4_8IOL:C.Data[116].1   // IO-Link Port 7 - Cycle time (ENUM bit1): 01001010=10.4 ms, 01001100=11.2 ms, 01001110=12.0 ms, 01010000=12.8 ms, 01010100=14.4 ms, 01011000=16.0 ms, 01011100=17.6 ms, 01100000=19.2 ms, 01100100=20.8 ms, 01101000=22.4 ms, 01101100=24.0 ms, 01110000=25.6 ms
           TBEN_L4_8IOL:C.Data[116].2   // IO-Link Port 7 - Cycle time (ENUM bit2): 01110100=27.2 ms, 01111000=28.8 ms, 01111100=30.4 ms, 10000000=32.0 ms, 10000001=33.6 ms, 10000010=35.2 ms, 10000011=36.8 ms, 10000100=38.4 ms, 10000101=40.0 ms, 10000110=41.6 ms, 10000111=43.2 ms, 10001000=44.8 ms
           TBEN_L4_8IOL:C.Data[116].3   // IO-Link Port 7 - Cycle time (ENUM bit3): 10001001=46.4 ms, 10001010=48.0 ms, 10001011=49.6 ms, 10001100=51.2 ms, 10001101=52.8 ms, 10001110=54.4 ms, 10001111=56.0 ms, 10010000=57.6 ms, 10010001=59.2 ms, 10010010=60.8 ms, 10010011=62.4 ms, 10010100=64.0 ms
           TBEN_L4_8IOL:C.Data[116].4   // IO-Link Port 7 - Cycle time (ENUM bit4): 10010101=65.6 ms, 10010110=67.2 ms, 10010111=68.8 ms, 10011000=70.4 ms, 10011001=72.0 ms, 10011010=73.6 ms, 10011011=75.2 ms, 10011100=76.8 ms, 10011101=78.4 ms, 10011110=80.0 ms, 10011111=81.6 ms
           TBEN_L4_8IOL:C.Data[116].5   // IO-Link Port 7 - Cycle time (ENUM bit5): 10100000=83.2 ms, 10100001=84.8 ms, 10100010=86.4 ms, 10100011=88.0 ms, 10100100=89.6 ms, 10100101=91.2 ms, 10100110=92.8 ms, 10100111=94.4 ms, 10101000=96.0 ms, 10101001=97.6 ms, 10101010=99.2 ms
           TBEN_L4_8IOL:C.Data[116].6   // IO-Link Port 7 - Cycle time (ENUM bit6): 10101011=100.8 ms, 10101100=102.4 ms, 10101101=104.0 ms, 10101110=105.6 ms, 10101111=107.2 ms, 10110000=108.8 ms, 10110001=110.4 ms, 10110010=112.0 ms, 10110011=113.6 ms, 10110100=115.2 ms, 10110101=116.8 ms
           TBEN_L4_8IOL:C.Data[116].7   // IO-Link Port 7 - Cycle time (ENUM bit7): 10110110=118.4 ms, 10110111=120.0 ms, 10111000=121.6 ms, 10111001=123.2 ms, 10111010=124.8 ms, 10111011=126.4 ms, 10111100=128.0 ms, 10111101=129.6 ms, 10111110=131.2 ms, 10111111=132.8 ms, 11111111=automatic, compatible
           TBEN_L4_8IOL:C.Data[117]   // IO-Link Port 7 - Revision
           TBEN_L4_8IOL:C.Data[117].0   // IO-Link Port 7 - Revision (ENUM bit0): 0=automatic, 1=V1.0
           TBEN_L4_8IOL:C.Data[117].1   // Reserved
           TBEN_L4_8IOL:C.Data[117].2   // Reserved
           TBEN_L4_8IOL:C.Data[117].3   // Reserved
           TBEN_L4_8IOL:C.Data[117].4   // Reserved
           TBEN_L4_8IOL:C.Data[117].5   // Reserved
           TBEN_L4_8IOL:C.Data[117].6   // Reserved
           TBEN_L4_8IOL:C.Data[117].7   // Reserved
           TBEN_L4_8IOL:C.Data[118]   // IO-Link Port 7 - Activate Quick Start-Up
           TBEN_L4_8IOL:C.Data[118].0   // IO-Link Port 7 - Activate Quick Start-Up (ENUM bit0): 0=no, 1=yes
           TBEN_L4_8IOL:C.Data[118].1   // Reserved
           TBEN_L4_8IOL:C.Data[118].2   // Reserved
           TBEN_L4_8IOL:C.Data[118].3   // Reserved
           TBEN_L4_8IOL:C.Data[118].4   // Reserved
           TBEN_L4_8IOL:C.Data[118].5   // Reserved
           TBEN_L4_8IOL:C.Data[118].6   // Reserved
           TBEN_L4_8IOL:C.Data[118].7   // Reserved
           TBEN_L4_8IOL:C.Data[119]   // IO-Link Port 7 - Device parametrization via GSD
           TBEN_L4_8IOL:C.Data[119].0   // IO-Link Port 7 - Device parametrization via GSD (ENUM bit0): 0=inactive, 1=active
           TBEN_L4_8IOL:C.Data[119].1   // Reserved
           TBEN_L4_8IOL:C.Data[119].2   // Reserved
           TBEN_L4_8IOL:C.Data[119].3   // Reserved
           TBEN_L4_8IOL:C.Data[119].4   // Reserved
           TBEN_L4_8IOL:C.Data[119].5   // Reserved
           TBEN_L4_8IOL:C.Data[119].6   // Reserved
           TBEN_L4_8IOL:C.Data[119].7   // Reserved
           TBEN_L4_8IOL:C.Data[11]   // DXP 3 - Manual reset after overcurr.
           TBEN_L4_8IOL:C.Data[11].0   // DXP 3 - Manual reset after overcurr. (ENUM bit0): 0=no, 1=yes
           TBEN_L4_8IOL:C.Data[11].1   // Reserved
           TBEN_L4_8IOL:C.Data[11].2   // Reserved
           TBEN_L4_8IOL:C.Data[11].3   // Reserved
           TBEN_L4_8IOL:C.Data[11].4   // Reserved
           TBEN_L4_8IOL:C.Data[11].5   // Reserved
           TBEN_L4_8IOL:C.Data[11].6   // Reserved
           TBEN_L4_8IOL:C.Data[11].7   // Reserved
           TBEN_L4_8IOL:C.Data[120]   // IO-Link Port 7 - Process input data invalid
           TBEN_L4_8IOL:C.Data[120].0   // IO-Link Port 7 - Process input data invalid (ENUM bit0): 0=diagnostic generated, 1=no diagnostic generated
           TBEN_L4_8IOL:C.Data[120].1   // Reserved
           TBEN_L4_8IOL:C.Data[120].2   // Reserved
           TBEN_L4_8IOL:C.Data[120].3   // Reserved
           TBEN_L4_8IOL:C.Data[120].4   // Reserved
           TBEN_L4_8IOL:C.Data[120].5   // Reserved
           TBEN_L4_8IOL:C.Data[120].6   // Reserved
           TBEN_L4_8IOL:C.Data[120].7   // Reserved
           TBEN_L4_8IOL:C.Data[121]   // IO-Link Port 7 - Deactivate diagnostics
           TBEN_L4_8IOL:C.Data[121].0   // IO-Link Port 7 - Deactivate diagnostics (ENUM bit0): 00=no, 01=notifications
           TBEN_L4_8IOL:C.Data[121].1   // IO-Link Port 7 - Deactivate diagnostics (ENUM bit1): 10=notifications and warnings, 11=yes
           TBEN_L4_8IOL:C.Data[121].2   // Reserved
           TBEN_L4_8IOL:C.Data[121].3   // Reserved
           TBEN_L4_8IOL:C.Data[121].4   // Reserved
           TBEN_L4_8IOL:C.Data[121].5   // Reserved
           TBEN_L4_8IOL:C.Data[121].6   // Reserved
           TBEN_L4_8IOL:C.Data[121].7   // Reserved
           TBEN_L4_8IOL:C.Data[122]   // IO-Link Port 7 - Input data mapping
           TBEN_L4_8IOL:C.Data[122].0   // IO-Link Port 7 - Input data mapping (ENUM bit0): 00=direct, 01=swap 16 bit
           TBEN_L4_8IOL:C.Data[122].1   // IO-Link Port 7 - Input data mapping (ENUM bit1): 10=swap 32 bit, 11=swap
           TBEN_L4_8IOL:C.Data[122].2   // Reserved
           TBEN_L4_8IOL:C.Data[122].3   // Reserved
           TBEN_L4_8IOL:C.Data[122].4   // Reserved
           TBEN_L4_8IOL:C.Data[122].5   // Reserved
           TBEN_L4_8IOL:C.Data[122].6   // Reserved
           TBEN_L4_8IOL:C.Data[122].7   // Reserved
           TBEN_L4_8IOL:C.Data[123]   // IO-Link Port 7 - Output data mapping
           TBEN_L4_8IOL:C.Data[123].0   // IO-Link Port 7 - Output data mapping (ENUM bit0): 00=direct, 01=swap 16 bit
           TBEN_L4_8IOL:C.Data[123].1   // IO-Link Port 7 - Output data mapping (ENUM bit1): 10=swap 32 bit, 11=swap
           TBEN_L4_8IOL:C.Data[123].2   // Reserved
           TBEN_L4_8IOL:C.Data[123].3   // Reserved
           TBEN_L4_8IOL:C.Data[123].4   // Reserved
           TBEN_L4_8IOL:C.Data[123].5   // Reserved
           TBEN_L4_8IOL:C.Data[123].6   // Reserved
           TBEN_L4_8IOL:C.Data[123].7   // Reserved
           TBEN_L4_8IOL:C.Data[124]   // IO-Link Port 7 - Vendor ID
           TBEN_L4_8IOL:C.Data[124].0   // IO-Link Port 7 - Vendor ID (INT bit0)
           TBEN_L4_8IOL:C.Data[124].1   // IO-Link Port 7 - Vendor ID (INT bit1)
           TBEN_L4_8IOL:C.Data[124].2   // IO-Link Port 7 - Vendor ID (INT bit2)
           TBEN_L4_8IOL:C.Data[124].3   // IO-Link Port 7 - Vendor ID (INT bit3)
           TBEN_L4_8IOL:C.Data[124].4   // IO-Link Port 7 - Vendor ID (INT bit4)
           TBEN_L4_8IOL:C.Data[124].5   // IO-Link Port 7 - Vendor ID (INT bit5)
           TBEN_L4_8IOL:C.Data[124].6   // IO-Link Port 7 - Vendor ID (INT bit6)
           TBEN_L4_8IOL:C.Data[124].7   // IO-Link Port 7 - Vendor ID (INT bit7)
           TBEN_L4_8IOL:C.Data[125]   // IO-Link Port 7 - Vendor ID
           TBEN_L4_8IOL:C.Data[125].0   // IO-Link Port 7 - Vendor ID (INT bit8)
           TBEN_L4_8IOL:C.Data[125].1   // IO-Link Port 7 - Vendor ID (INT bit9)
           TBEN_L4_8IOL:C.Data[125].2   // IO-Link Port 7 - Vendor ID (INT bit10)
           TBEN_L4_8IOL:C.Data[125].3   // IO-Link Port 7 - Vendor ID (INT bit11)
           TBEN_L4_8IOL:C.Data[125].4   // IO-Link Port 7 - Vendor ID (INT bit12)
           TBEN_L4_8IOL:C.Data[125].5   // IO-Link Port 7 - Vendor ID (INT bit13)
           TBEN_L4_8IOL:C.Data[125].6   // IO-Link Port 7 - Vendor ID (INT bit14)
           TBEN_L4_8IOL:C.Data[125].7   // IO-Link Port 7 - Vendor ID (INT bit15)
           TBEN_L4_8IOL:C.Data[126]   // IO-Link Port 7 - Device ID
           TBEN_L4_8IOL:C.Data[126].0   // IO-Link Port 7 - Device ID (INT bit0)
           TBEN_L4_8IOL:C.Data[126].1   // IO-Link Port 7 - Device ID (INT bit1)
           TBEN_L4_8IOL:C.Data[126].2   // IO-Link Port 7 - Device ID (INT bit2)
           TBEN_L4_8IOL:C.Data[126].3   // IO-Link Port 7 - Device ID (INT bit3)
           TBEN_L4_8IOL:C.Data[126].4   // IO-Link Port 7 - Device ID (INT bit4)
           TBEN_L4_8IOL:C.Data[126].5   // IO-Link Port 7 - Device ID (INT bit5)
           TBEN_L4_8IOL:C.Data[126].6   // IO-Link Port 7 - Device ID (INT bit6)
           TBEN_L4_8IOL:C.Data[126].7   // IO-Link Port 7 - Device ID (INT bit7)
           TBEN_L4_8IOL:C.Data[127]   // IO-Link Port 7 - Device ID
           TBEN_L4_8IOL:C.Data[127].0   // IO-Link Port 7 - Device ID (INT bit8)
           TBEN_L4_8IOL:C.Data[127].1   // IO-Link Port 7 - Device ID (INT bit9)
           TBEN_L4_8IOL:C.Data[127].2   // IO-Link Port 7 - Device ID (INT bit10)
           TBEN_L4_8IOL:C.Data[127].3   // IO-Link Port 7 - Device ID (INT bit11)
           TBEN_L4_8IOL:C.Data[127].4   // IO-Link Port 7 - Device ID (INT bit12)
           TBEN_L4_8IOL:C.Data[127].5   // IO-Link Port 7 - Device ID (INT bit13)
           TBEN_L4_8IOL:C.Data[127].6   // IO-Link Port 7 - Device ID (INT bit14)
           TBEN_L4_8IOL:C.Data[127].7   // IO-Link Port 7 - Device ID (INT bit15)
           TBEN_L4_8IOL:C.Data[128]   // IO-Link Port 7 - Device ID
           TBEN_L4_8IOL:C.Data[128].0   // IO-Link Port 7 - Device ID (INT bit16)
           TBEN_L4_8IOL:C.Data[128].1   // IO-Link Port 7 - Device ID (INT bit17)
           TBEN_L4_8IOL:C.Data[128].2   // IO-Link Port 7 - Device ID (INT bit18)
           TBEN_L4_8IOL:C.Data[128].3   // IO-Link Port 7 - Device ID (INT bit19)
           TBEN_L4_8IOL:C.Data[128].4   // IO-Link Port 7 - Device ID (INT bit20)
           TBEN_L4_8IOL:C.Data[128].5   // IO-Link Port 7 - Device ID (INT bit21)
           TBEN_L4_8IOL:C.Data[128].6   // IO-Link Port 7 - Device ID (INT bit22)
           TBEN_L4_8IOL:C.Data[128].7   // IO-Link Port 7 - Device ID (INT bit23)
           TBEN_L4_8IOL:C.Data[129]   // IO-Link Port 7 - Device ID
           TBEN_L4_8IOL:C.Data[129].0   // IO-Link Port 7 - Device ID (INT bit24)
           TBEN_L4_8IOL:C.Data[129].1   // IO-Link Port 7 - Device ID (INT bit25)
           TBEN_L4_8IOL:C.Data[129].2   // IO-Link Port 7 - Device ID (INT bit26)
           TBEN_L4_8IOL:C.Data[129].3   // IO-Link Port 7 - Device ID (INT bit27)
           TBEN_L4_8IOL:C.Data[129].4   // IO-Link Port 7 - Device ID (INT bit28)
           TBEN_L4_8IOL:C.Data[129].5   // IO-Link Port 7 - Device ID (INT bit29)
           TBEN_L4_8IOL:C.Data[129].6   // IO-Link Port 7 - Device ID (INT bit30)
           TBEN_L4_8IOL:C.Data[129].7   // IO-Link Port 7 - Device ID (INT bit31)
           TBEN_L4_8IOL:C.Data[12]   // DXP 5 - Manual reset after overcurr.
           TBEN_L4_8IOL:C.Data[12].0   // DXP 5 - Manual reset after overcurr. (ENUM bit0): 0=no, 1=yes
           TBEN_L4_8IOL:C.Data[12].1   // Reserved
           TBEN_L4_8IOL:C.Data[12].2   // Reserved
           TBEN_L4_8IOL:C.Data[12].3   // Reserved
           TBEN_L4_8IOL:C.Data[12].4   // Reserved
           TBEN_L4_8IOL:C.Data[12].5   // Reserved
           TBEN_L4_8IOL:C.Data[12].6   // Reserved
           TBEN_L4_8IOL:C.Data[12].7   // Reserved
           TBEN_L4_8IOL:C.Data[130]   // IO-Link Port 8 - Operation mode
           TBEN_L4_8IOL:C.Data[130].0   // IO-Link Port 8 - Operation mode (ENUM bit0): 0000=IO-Link without validation, 0001=IO-Link with family compatible device
           TBEN_L4_8IOL:C.Data[130].1   // IO-Link Port 8 - Operation mode (ENUM bit1): 0010=IO-Link with compatible device, 0011=IO-Link with identical device
           TBEN_L4_8IOL:C.Data[130].2   // IO-Link Port 8 - Operation mode (ENUM bit2): 0100=DI (with parameter access)
           TBEN_L4_8IOL:C.Data[130].3   // IO-Link Port 8 - Operation mode (ENUM bit3): 1000=DI
           TBEN_L4_8IOL:C.Data[130].4   // Reserved
           TBEN_L4_8IOL:C.Data[130].5   // Reserved
           TBEN_L4_8IOL:C.Data[130].6   // Reserved
           TBEN_L4_8IOL:C.Data[130].7   // Reserved
           TBEN_L4_8IOL:C.Data[131]   // IO-Link Port 8 - Data storage mode
           TBEN_L4_8IOL:C.Data[131].0   // IO-Link Port 8 - Data storage mode (ENUM bit0): 00=activated, 01=overwrite
           TBEN_L4_8IOL:C.Data[131].1   // IO-Link Port 8 - Data storage mode (ENUM bit1): 10=read in, 11=deactivated, clear
           TBEN_L4_8IOL:C.Data[131].2   // Reserved
           TBEN_L4_8IOL:C.Data[131].3   // Reserved
           TBEN_L4_8IOL:C.Data[131].4   // Reserved
           TBEN_L4_8IOL:C.Data[131].5   // Reserved
           TBEN_L4_8IOL:C.Data[131].6   // Reserved
           TBEN_L4_8IOL:C.Data[131].7   // Reserved
           TBEN_L4_8IOL:C.Data[132]   // IO-Link Port 8 - Cycle time
           TBEN_L4_8IOL:C.Data[132].0   // IO-Link Port 8 - Cycle time (ENUM bit0): 00000000=automatic, 00010000=1.6 ms, 00011000=2.4 ms, 00100000=3.2 ms, 00101000=4.0 ms, 00110000=4.8 ms, 00111000=5.6 ms, 01000000=6.4 ms, 01000010=7.2 ms, 01000100=8.0 ms, 01000110=8.8 ms, 01001000=9.6 ms
           TBEN_L4_8IOL:C.Data[132].1   // IO-Link Port 8 - Cycle time (ENUM bit1): 01001010=10.4 ms, 01001100=11.2 ms, 01001110=12.0 ms, 01010000=12.8 ms, 01010100=14.4 ms, 01011000=16.0 ms, 01011100=17.6 ms, 01100000=19.2 ms, 01100100=20.8 ms, 01101000=22.4 ms, 01101100=24.0 ms, 01110000=25.6 ms
           TBEN_L4_8IOL:C.Data[132].2   // IO-Link Port 8 - Cycle time (ENUM bit2): 01110100=27.2 ms, 01111000=28.8 ms, 01111100=30.4 ms, 10000000=32.0 ms, 10000001=33.6 ms, 10000010=35.2 ms, 10000011=36.8 ms, 10000100=38.4 ms, 10000101=40.0 ms, 10000110=41.6 ms, 10000111=43.2 ms, 10001000=44.8 ms
           TBEN_L4_8IOL:C.Data[132].3   // IO-Link Port 8 - Cycle time (ENUM bit3): 10001001=46.4 ms, 10001010=48.0 ms, 10001011=49.6 ms, 10001100=51.2 ms, 10001101=52.8 ms, 10001110=54.4 ms, 10001111=56.0 ms, 10010000=57.6 ms, 10010001=59.2 ms, 10010010=60.8 ms, 10010011=62.4 ms, 10010100=64.0 ms
           TBEN_L4_8IOL:C.Data[132].4   // IO-Link Port 8 - Cycle time (ENUM bit4): 10010101=65.6 ms, 10010110=67.2 ms, 10010111=68.8 ms, 10011000=70.4 ms, 10011001=72.0 ms, 10011010=73.6 ms, 10011011=75.2 ms, 10011100=76.8 ms, 10011101=78.4 ms, 10011110=80.0 ms, 10011111=81.6 ms
           TBEN_L4_8IOL:C.Data[132].5   // IO-Link Port 8 - Cycle time (ENUM bit5): 10100000=83.2 ms, 10100001=84.8 ms, 10100010=86.4 ms, 10100011=88.0 ms, 10100100=89.6 ms, 10100101=91.2 ms, 10100110=92.8 ms, 10100111=94.4 ms, 10101000=96.0 ms, 10101001=97.6 ms, 10101010=99.2 ms
           TBEN_L4_8IOL:C.Data[132].6   // IO-Link Port 8 - Cycle time (ENUM bit6): 10101011=100.8 ms, 10101100=102.4 ms, 10101101=104.0 ms, 10101110=105.6 ms, 10101111=107.2 ms, 10110000=108.8 ms, 10110001=110.4 ms, 10110010=112.0 ms, 10110011=113.6 ms, 10110100=115.2 ms, 10110101=116.8 ms
           TBEN_L4_8IOL:C.Data[132].7   // IO-Link Port 8 - Cycle time (ENUM bit7): 10110110=118.4 ms, 10110111=120.0 ms, 10111000=121.6 ms, 10111001=123.2 ms, 10111010=124.8 ms, 10111011=126.4 ms, 10111100=128.0 ms, 10111101=129.6 ms, 10111110=131.2 ms, 10111111=132.8 ms, 11111111=automatic, compatible
           TBEN_L4_8IOL:C.Data[133]   // IO-Link Port 8 - Revision
           TBEN_L4_8IOL:C.Data[133].0   // IO-Link Port 8 - Revision (ENUM bit0): 0=automatic, 1=V1.0
           TBEN_L4_8IOL:C.Data[133].1   // Reserved
           TBEN_L4_8IOL:C.Data[133].2   // Reserved
           TBEN_L4_8IOL:C.Data[133].3   // Reserved
           TBEN_L4_8IOL:C.Data[133].4   // Reserved
           TBEN_L4_8IOL:C.Data[133].5   // Reserved
           TBEN_L4_8IOL:C.Data[133].6   // Reserved
           TBEN_L4_8IOL:C.Data[133].7   // Reserved
           TBEN_L4_8IOL:C.Data[134]   // IO-Link Port 8 - Activate Quick Start-Up
           TBEN_L4_8IOL:C.Data[134].0   // IO-Link Port 8 - Activate Quick Start-Up (ENUM bit0): 0=no, 1=yes
           TBEN_L4_8IOL:C.Data[134].1   // Reserved
           TBEN_L4_8IOL:C.Data[134].2   // Reserved
           TBEN_L4_8IOL:C.Data[134].3   // Reserved
           TBEN_L4_8IOL:C.Data[134].4   // Reserved
           TBEN_L4_8IOL:C.Data[134].5   // Reserved
           TBEN_L4_8IOL:C.Data[134].6   // Reserved
           TBEN_L4_8IOL:C.Data[134].7   // Reserved
           TBEN_L4_8IOL:C.Data[135]   // IO-Link Port 8 - Device parametrization via GSD
           TBEN_L4_8IOL:C.Data[135].0   // IO-Link Port 8 - Device parametrization via GSD (ENUM bit0): 0=inactive, 1=active
           TBEN_L4_8IOL:C.Data[135].1   // Reserved
           TBEN_L4_8IOL:C.Data[135].2   // Reserved
           TBEN_L4_8IOL:C.Data[135].3   // Reserved
           TBEN_L4_8IOL:C.Data[135].4   // Reserved
           TBEN_L4_8IOL:C.Data[135].5   // Reserved
           TBEN_L4_8IOL:C.Data[135].6   // Reserved
           TBEN_L4_8IOL:C.Data[135].7   // Reserved
           TBEN_L4_8IOL:C.Data[136]   // IO-Link Port 8 - Process input data invalid
           TBEN_L4_8IOL:C.Data[136].0   // IO-Link Port 8 - Process input data invalid (ENUM bit0): 0=diagnostic generated, 1=no diagnostic generated
           TBEN_L4_8IOL:C.Data[136].1   // Reserved
           TBEN_L4_8IOL:C.Data[136].2   // Reserved
           TBEN_L4_8IOL:C.Data[136].3   // Reserved
           TBEN_L4_8IOL:C.Data[136].4   // Reserved
           TBEN_L4_8IOL:C.Data[136].5   // Reserved
           TBEN_L4_8IOL:C.Data[136].6   // Reserved
           TBEN_L4_8IOL:C.Data[136].7   // Reserved
           TBEN_L4_8IOL:C.Data[137]   // IO-Link Port 8 - Deactivate diagnostics
           TBEN_L4_8IOL:C.Data[137].0   // IO-Link Port 8 - Deactivate diagnostics (ENUM bit0): 00=no, 01=notifications
           TBEN_L4_8IOL:C.Data[137].1   // IO-Link Port 8 - Deactivate diagnostics (ENUM bit1): 10=notifications and warnings, 11=yes
           TBEN_L4_8IOL:C.Data[137].2   // Reserved
           TBEN_L4_8IOL:C.Data[137].3   // Reserved
           TBEN_L4_8IOL:C.Data[137].4   // Reserved
           TBEN_L4_8IOL:C.Data[137].5   // Reserved
           TBEN_L4_8IOL:C.Data[137].6   // Reserved
           TBEN_L4_8IOL:C.Data[137].7   // Reserved
           TBEN_L4_8IOL:C.Data[138]   // IO-Link Port 8 - Input data mapping
           TBEN_L4_8IOL:C.Data[138].0   // IO-Link Port 8 - Input data mapping (ENUM bit0): 00=direct, 01=swap 16 bit
           TBEN_L4_8IOL:C.Data[138].1   // IO-Link Port 8 - Input data mapping (ENUM bit1): 10=swap 32 bit, 11=swap
           TBEN_L4_8IOL:C.Data[138].2   // Reserved
           TBEN_L4_8IOL:C.Data[138].3   // Reserved
           TBEN_L4_8IOL:C.Data[138].4   // Reserved
           TBEN_L4_8IOL:C.Data[138].5   // Reserved
           TBEN_L4_8IOL:C.Data[138].6   // Reserved
           TBEN_L4_8IOL:C.Data[138].7   // Reserved
           TBEN_L4_8IOL:C.Data[139]   // IO-Link Port 8 - Output data mapping
           TBEN_L4_8IOL:C.Data[139].0   // IO-Link Port 8 - Output data mapping (ENUM bit0): 00=direct, 01=swap 16 bit
           TBEN_L4_8IOL:C.Data[139].1   // IO-Link Port 8 - Output data mapping (ENUM bit1): 10=swap 32 bit, 11=swap
           TBEN_L4_8IOL:C.Data[139].2   // Reserved
           TBEN_L4_8IOL:C.Data[139].3   // Reserved
           TBEN_L4_8IOL:C.Data[139].4   // Reserved
           TBEN_L4_8IOL:C.Data[139].5   // Reserved
           TBEN_L4_8IOL:C.Data[139].6   // Reserved
           TBEN_L4_8IOL:C.Data[139].7   // Reserved
           TBEN_L4_8IOL:C.Data[13]   // DXP 7 - Manual reset after overcurr.
           TBEN_L4_8IOL:C.Data[13].0   // DXP 7 - Manual reset after overcurr. (ENUM bit0): 0=no, 1=yes
           TBEN_L4_8IOL:C.Data[13].1   // Reserved
           TBEN_L4_8IOL:C.Data[13].2   // Reserved
           TBEN_L4_8IOL:C.Data[13].3   // Reserved
           TBEN_L4_8IOL:C.Data[13].4   // Reserved
           TBEN_L4_8IOL:C.Data[13].5   // Reserved
           TBEN_L4_8IOL:C.Data[13].6   // Reserved
           TBEN_L4_8IOL:C.Data[13].7   // Reserved
           TBEN_L4_8IOL:C.Data[140]   // IO-Link Port 8 - Vendor ID
           TBEN_L4_8IOL:C.Data[140].0   // IO-Link Port 8 - Vendor ID (INT bit0)
           TBEN_L4_8IOL:C.Data[140].1   // IO-Link Port 8 - Vendor ID (INT bit1)
           TBEN_L4_8IOL:C.Data[140].2   // IO-Link Port 8 - Vendor ID (INT bit2)
           TBEN_L4_8IOL:C.Data[140].3   // IO-Link Port 8 - Vendor ID (INT bit3)
           TBEN_L4_8IOL:C.Data[140].4   // IO-Link Port 8 - Vendor ID (INT bit4)
           TBEN_L4_8IOL:C.Data[140].5   // IO-Link Port 8 - Vendor ID (INT bit5)
           TBEN_L4_8IOL:C.Data[140].6   // IO-Link Port 8 - Vendor ID (INT bit6)
           TBEN_L4_8IOL:C.Data[140].7   // IO-Link Port 8 - Vendor ID (INT bit7)
           TBEN_L4_8IOL:C.Data[141]   // IO-Link Port 8 - Vendor ID
           TBEN_L4_8IOL:C.Data[141].0   // IO-Link Port 8 - Vendor ID (INT bit8)
           TBEN_L4_8IOL:C.Data[141].1   // IO-Link Port 8 - Vendor ID (INT bit9)
           TBEN_L4_8IOL:C.Data[141].2   // IO-Link Port 8 - Vendor ID (INT bit10)
           TBEN_L4_8IOL:C.Data[141].3   // IO-Link Port 8 - Vendor ID (INT bit11)
           TBEN_L4_8IOL:C.Data[141].4   // IO-Link Port 8 - Vendor ID (INT bit12)
           TBEN_L4_8IOL:C.Data[141].5   // IO-Link Port 8 - Vendor ID (INT bit13)
           TBEN_L4_8IOL:C.Data[141].6   // IO-Link Port 8 - Vendor ID (INT bit14)
           TBEN_L4_8IOL:C.Data[141].7   // IO-Link Port 8 - Vendor ID (INT bit15)
           TBEN_L4_8IOL:C.Data[142]   // IO-Link Port 8 - Device ID
           TBEN_L4_8IOL:C.Data[142].0   // IO-Link Port 8 - Device ID (INT bit0)
           TBEN_L4_8IOL:C.Data[142].1   // IO-Link Port 8 - Device ID (INT bit1)
           TBEN_L4_8IOL:C.Data[142].2   // IO-Link Port 8 - Device ID (INT bit2)
           TBEN_L4_8IOL:C.Data[142].3   // IO-Link Port 8 - Device ID (INT bit3)
           TBEN_L4_8IOL:C.Data[142].4   // IO-Link Port 8 - Device ID (INT bit4)
           TBEN_L4_8IOL:C.Data[142].5   // IO-Link Port 8 - Device ID (INT bit5)
           TBEN_L4_8IOL:C.Data[142].6   // IO-Link Port 8 - Device ID (INT bit6)
           TBEN_L4_8IOL:C.Data[142].7   // IO-Link Port 8 - Device ID (INT bit7)
           TBEN_L4_8IOL:C.Data[143]   // IO-Link Port 8 - Device ID
           TBEN_L4_8IOL:C.Data[143].0   // IO-Link Port 8 - Device ID (INT bit8)
           TBEN_L4_8IOL:C.Data[143].1   // IO-Link Port 8 - Device ID (INT bit9)
           TBEN_L4_8IOL:C.Data[143].2   // IO-Link Port 8 - Device ID (INT bit10)
           TBEN_L4_8IOL:C.Data[143].3   // IO-Link Port 8 - Device ID (INT bit11)
           TBEN_L4_8IOL:C.Data[143].4   // IO-Link Port 8 - Device ID (INT bit12)
           TBEN_L4_8IOL:C.Data[143].5   // IO-Link Port 8 - Device ID (INT bit13)
           TBEN_L4_8IOL:C.Data[143].6   // IO-Link Port 8 - Device ID (INT bit14)
           TBEN_L4_8IOL:C.Data[143].7   // IO-Link Port 8 - Device ID (INT bit15)
           TBEN_L4_8IOL:C.Data[144]   // IO-Link Port 8 - Device ID
           TBEN_L4_8IOL:C.Data[144].0   // IO-Link Port 8 - Device ID (INT bit16)
           TBEN_L4_8IOL:C.Data[144].1   // IO-Link Port 8 - Device ID (INT bit17)
           TBEN_L4_8IOL:C.Data[144].2   // IO-Link Port 8 - Device ID (INT bit18)
           TBEN_L4_8IOL:C.Data[144].3   // IO-Link Port 8 - Device ID (INT bit19)
           TBEN_L4_8IOL:C.Data[144].4   // IO-Link Port 8 - Device ID (INT bit20)
           TBEN_L4_8IOL:C.Data[144].5   // IO-Link Port 8 - Device ID (INT bit21)
